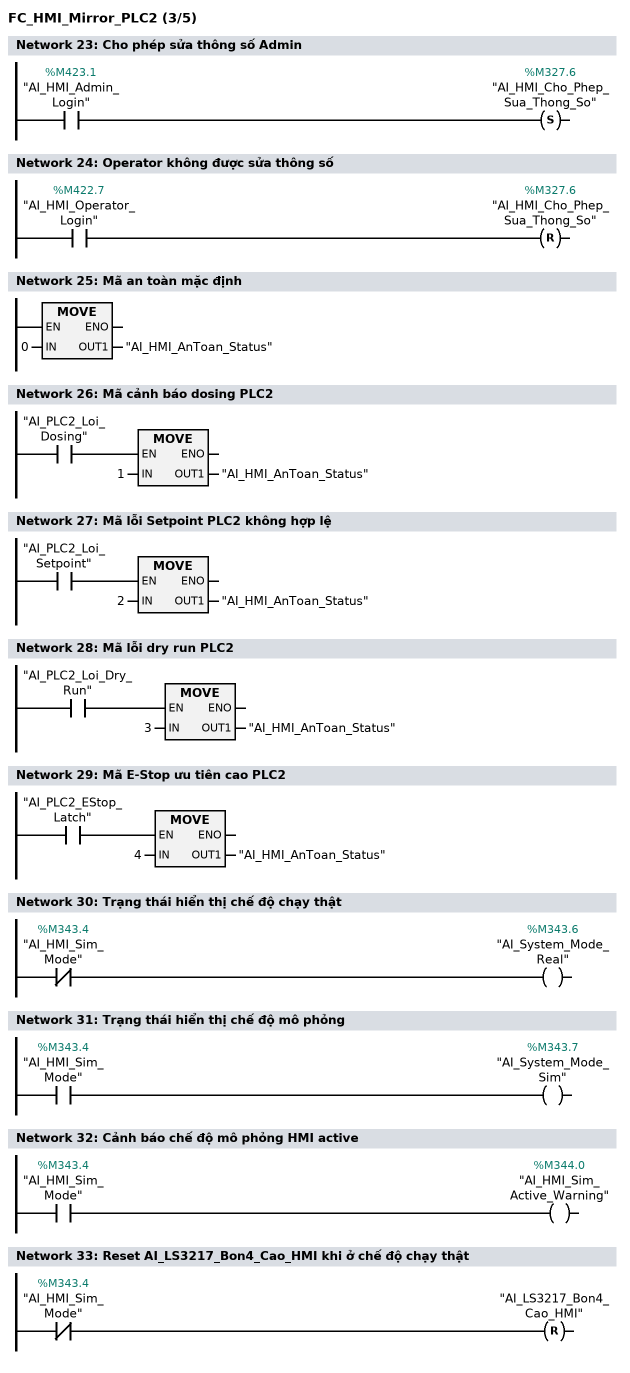
   RUNG wire#powerrail
      Contact( "AI_HMI_Admin_Login" )
      S_Coil( "AI_HMI_Cho_Phep_Sua_Thong_So" )
   END_RUNG
   // the same network as SCL:
   IF "AI_HMI_Admin_Login" THEN "AI_HMI_Cho_Phep_Sua_Thong_So" := TRUE; END_IF;
END_REGION

REGION Network 24: Operator không được sửa thông số
   RUNG wire#powerrail
      Contact( "AI_HMI_Operator_Login" )
      R_Coil( "AI_HMI_Cho_Phep_Sua_Thong_So" )
   END_RUNG
   // the same network as SCL:
   IF "AI_HMI_Operator_Login" THEN "AI_HMI_Cho_Phep_Sua_Thong_So" := FALSE; END_IF;
END_REGION

REGION Network 25: Mã an toàn mặc định
   RUNG wire#powerrail
      { S7_GenerateENO := "TRUE" } Move(in := 0, out1 => "AI_HMI_AnToan_Status")
   END_RUNG
   // the same network as SCL:
   "AI_HMI_AnToan_Status" := 0;
END_REGION

REGION Network 26: Mã cảnh báo dosing PLC2
   RUNG wire#powerrail
      Contact( "AI_PLC2_Loi_Dosing" )
      { S7_GenerateENO := "TRUE" } Move(in := 1, out1 => "AI_HMI_AnToan_Status")
   END_RUNG
   // the same network as SCL:
   IF "AI_PLC2_Loi_Dosing" THEN "AI_HMI_AnToan_Status" := 1; END_IF;
END_REGION

REGION Network 27: Mã lỗi Setpoint PLC2 không hợp lệ
   RUNG wire#powerrail
      Contact( "AI_PLC2_Loi_Setpoint" )
      { S7_GenerateENO := "TRUE" } Move(in := 2, out1 => "AI_HMI_AnToan_Status")
   END_RUNG
   // the same network as SCL:
   IF "AI_PLC2_Loi_Setpoint" THEN "AI_HMI_AnToan_Status" := 2; END_IF;
END_REGION

REGION Network 28: Mã lỗi dry run PLC2
   RUNG wire#powerrail
      Contact( "AI_PLC2_Loi_Dry_Run" )
      { S7_GenerateENO := "TRUE" } Move(in := 3, out1 => "AI_HMI_AnToan_Status")
   END_RUNG
   // the same network as SCL:
   IF "AI_PLC2_Loi_Dry_Run" THEN "AI_HMI_AnToan_Status" := 3; END_IF;
END_REGION

REGION Network 29: Mã E-Stop ưu tiên cao PLC2
   RUNG wire#powerrail
      Contact( "AI_PLC2_EStop_Latch" )
      { S7_GenerateENO := "TRUE" } Move(in := 4, out1 => "AI_HMI_AnToan_Status")
   END_RUNG
   // the same network as SCL:
   IF "AI_PLC2_EStop_Latch" THEN "AI_HMI_AnToan_Status" := 4; END_IF;
END_REGION

REGION Network 30: Trạng thái hiển thị chế độ chạy thật
   RUNG wire#powerrail
      I_Contact( "AI_HMI_Sim_Mode" )
      Coil( "AI_System_Mode_Real" )
   END_RUNG
   // the same network as SCL:
   "AI_System_Mode_Real" := NOT "AI_HMI_Sim_Mode";
END_REGION

REGION Network 31: Trạng thái hiển thị chế độ mô phỏng
   RUNG wire#powerrail
      Contact( "AI_HMI_Sim_Mode" )
      Coil( "AI_System_Mode_Sim" )
   END_RUNG
   // the same network as SCL:
   "AI_System_Mode_Sim" := "AI_HMI_Sim_Mode";
END_REGION

REGION Network 32: Cảnh báo chế độ mô phỏng HMI active
   RUNG wire#powerrail
      Contact( "AI_HMI_Sim_Mode" )
      Coil( "AI_HMI_Sim_Active_Warning" )
   END_RUNG
   // the same network as SCL:
   "AI_HMI_Sim_Active_Warning" := "AI_HMI_Sim_Mode";
END_REGION

REGION Network 33: Reset AI_LS3217_Bon4_Cao_HMI khi ở chế độ chạy thật
   RUNG wire#powerrail
      I_Contact( "AI_HMI_Sim_Mode" )
      R_Coil( "AI_LS3217_Bon4_Cao_HMI" )
   END_RUNG
   // the same network as SCL:
   IF NOT "AI_HMI_Sim_Mode" THEN "AI_LS3217_Bon4_Cao_HMI" := FALSE; END_IF;
END_REGION

REGION Network 34: Reset AI_Pump3265_Chuyen_Nhanh2_Cmd_Nhan_HMI khi ở chế độ chạy thật
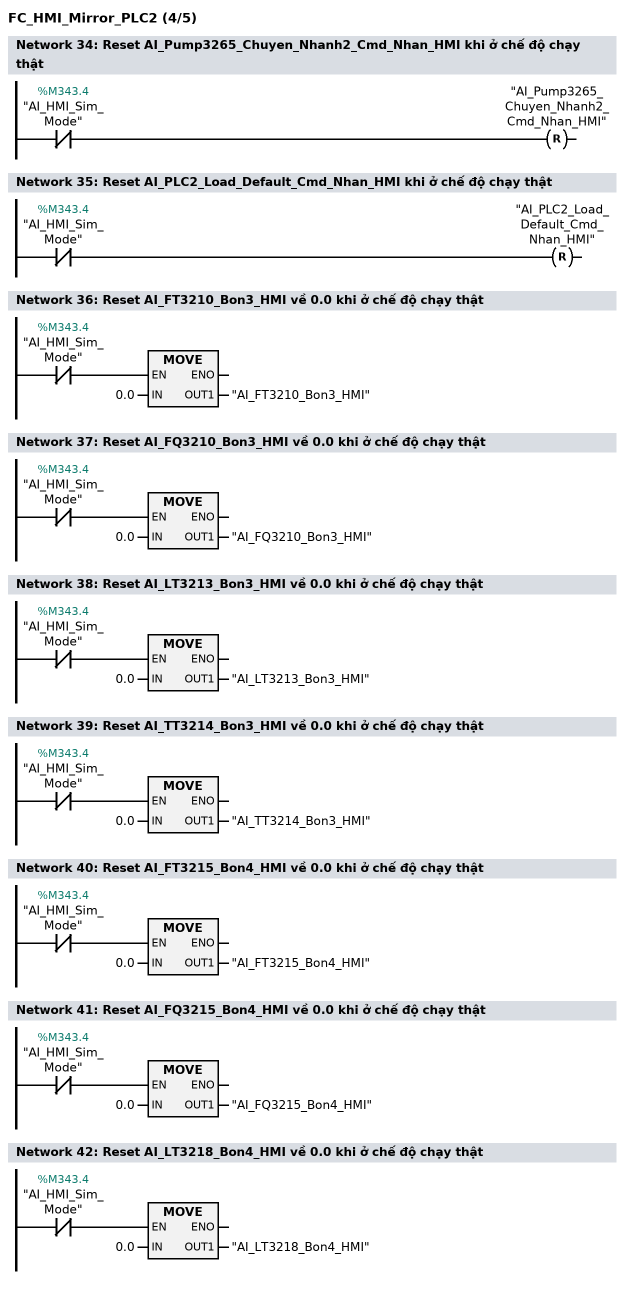
   RUNG wire#powerrail
      I_Contact( "AI_HMI_Sim_Mode" )
      R_Coil( "AI_Pump3265_Chuyen_Nhanh2_Cmd_Nhan_HMI" )
   END_RUNG
   // the same network as SCL:
   IF NOT "AI_HMI_Sim_Mode" THEN "AI_Pump3265_Chuyen_Nhanh2_Cmd_Nhan_HMI" := FALSE; END_IF;
END_REGION

REGION Network 35: Reset AI_PLC2_Load_Default_Cmd_Nhan_HMI khi ở chế độ chạy thật
   RUNG wire#powerrail
      I_Contact( "AI_HMI_Sim_Mode" )
      R_Coil( "AI_PLC2_Load_Default_Cmd_Nhan_HMI" )
   END_RUNG
   // the same network as SCL:
   IF NOT "AI_HMI_Sim_Mode" THEN "AI_PLC2_Load_Default_Cmd_Nhan_HMI" := FALSE; END_IF;
END_REGION

REGION Network 36: Reset AI_FT3210_Bon3_HMI về 0.0 khi ở chế độ chạy thật
   RUNG wire#powerrail
      I_Contact( "AI_HMI_Sim_Mode" )
      { S7_GenerateENO := "TRUE" } Move(in := 0.0, out1 => "AI_FT3210_Bon3_HMI")
   END_RUNG
   // the same network as SCL:
   IF NOT "AI_HMI_Sim_Mode" THEN "AI_FT3210_Bon3_HMI" := 0.0; END_IF;
END_REGION

REGION Network 37: Reset AI_FQ3210_Bon3_HMI về 0.0 khi ở chế độ chạy thật
   RUNG wire#powerrail
      I_Contact( "AI_HMI_Sim_Mode" )
      { S7_GenerateENO := "TRUE" } Move(in := 0.0, out1 => "AI_FQ3210_Bon3_HMI")
   END_RUNG
   // the same network as SCL:
   IF NOT "AI_HMI_Sim_Mode" THEN "AI_FQ3210_Bon3_HMI" := 0.0; END_IF;
END_REGION

REGION Network 38: Reset AI_LT3213_Bon3_HMI về 0.0 khi ở chế độ chạy thật
   RUNG wire#powerrail
      I_Contact( "AI_HMI_Sim_Mode" )
      { S7_GenerateENO := "TRUE" } Move(in := 0.0, out1 => "AI_LT3213_Bon3_HMI")
   END_RUNG
   // the same network as SCL:
   IF NOT "AI_HMI_Sim_Mode" THEN "AI_LT3213_Bon3_HMI" := 0.0; END_IF;
END_REGION

REGION Network 39: Reset AI_TT3214_Bon3_HMI về 0.0 khi ở chế độ chạy thật
   RUNG wire#powerrail
      I_Contact( "AI_HMI_Sim_Mode" )
      { S7_GenerateENO := "TRUE" } Move(in := 0.0, out1 => "AI_TT3214_Bon3_HMI")
   END_RUNG
   // the same network as SCL:
   IF NOT "AI_HMI_Sim_Mode" THEN "AI_TT3214_Bon3_HMI" := 0.0; END_IF;
END_REGION

REGION Network 40: Reset AI_FT3215_Bon4_HMI về 0.0 khi ở chế độ chạy thật
   RUNG wire#powerrail
      I_Contact( "AI_HMI_Sim_Mode" )
      { S7_GenerateENO := "TRUE" } Move(in := 0.0, out1 => "AI_FT3215_Bon4_HMI")
   END_RUNG
   // the same network as SCL:
   IF NOT "AI_HMI_Sim_Mode" THEN "AI_FT3215_Bon4_HMI" := 0.0; END_IF;
END_REGION

REGION Network 41: Reset AI_FQ3215_Bon4_HMI về 0.0 khi ở chế độ chạy thật
   RUNG wire#powerrail
      I_Contact( "AI_HMI_Sim_Mode" )
      { S7_GenerateENO := "TRUE" } Move(in := 0.0, out1 => "AI_FQ3215_Bon4_HMI")
   END_RUNG
   // the same network as SCL:
   IF NOT "AI_HMI_Sim_Mode" THEN "AI_FQ3215_Bon4_HMI" := 0.0; END_IF;
END_REGION

REGION Network 42: Reset AI_LT3218_Bon4_HMI về 0.0 khi ở chế độ chạy thật
   RUNG wire#powerrail
      I_Contact( "AI_HMI_Sim_Mode" )
      { S7_GenerateENO := "TRUE" } Move(in := 0.0, out1 => "AI_LT3218_Bon4_HMI")
   END_RUNG
   // the same network as SCL:
   IF NOT "AI_HMI_Sim_Mode" THEN "AI_LT3218_Bon4_HMI" := 0.0; END_IF;
END_REGION

REGION Network 43: Reset AI_TT3219_Bon4_HMI về 0.0 khi ở chế độ chạy thật
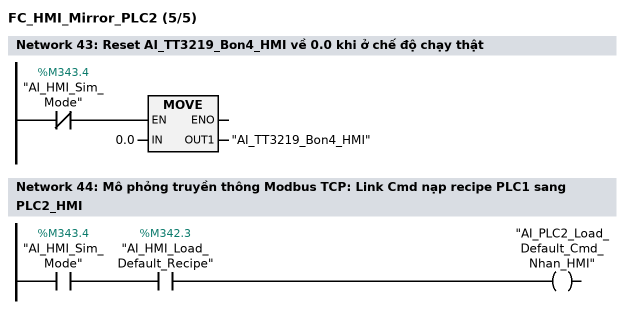
   RUNG wire#powerrail
      I_Contact( "AI_HMI_Sim_Mode" )
      { S7_GenerateENO := "TRUE" } Move(in := 0.0, out1 => "AI_TT3219_Bon4_HMI")
   END_RUNG
   // the same network as SCL:
   IF NOT "AI_HMI_Sim_Mode" THEN "AI_TT3219_Bon4_HMI" := 0.0; END_IF;
END_REGION

REGION Network 44: Mô phỏng truyền thông Modbus TCP: Link Cmd nạp recipe PLC1 sang PLC2_HMI
   RUNG wire#powerrail
      Contact( "AI_HMI_Sim_Mode" )
      Contact( "AI_HMI_Load_Default_Recipe" )
      Coil( "AI_PLC2_Load_Default_Cmd_Nhan_HMI" )
   END_RUNG
   // the same network as SCL:
   "AI_PLC2_Load_Default_Cmd_Nhan_HMI" := "AI_HMI_Sim_Mode" AND "AI_HMI_Load_Default_Recipe";
END_REGION
END_FUNCTION

FUNCTION "FC_Init_Default_Recipe_PLC2" : Void   // FC51, LAD
{ S7_Optimized_Access := 'TRUE' }
VERSION : 0.1
// stored: AutoNumber true, IsIECCheckEnabled false
BEGIN

REGION Network 1: Kích hoạt nạp recipe mặc định lần đầu scan PLC2
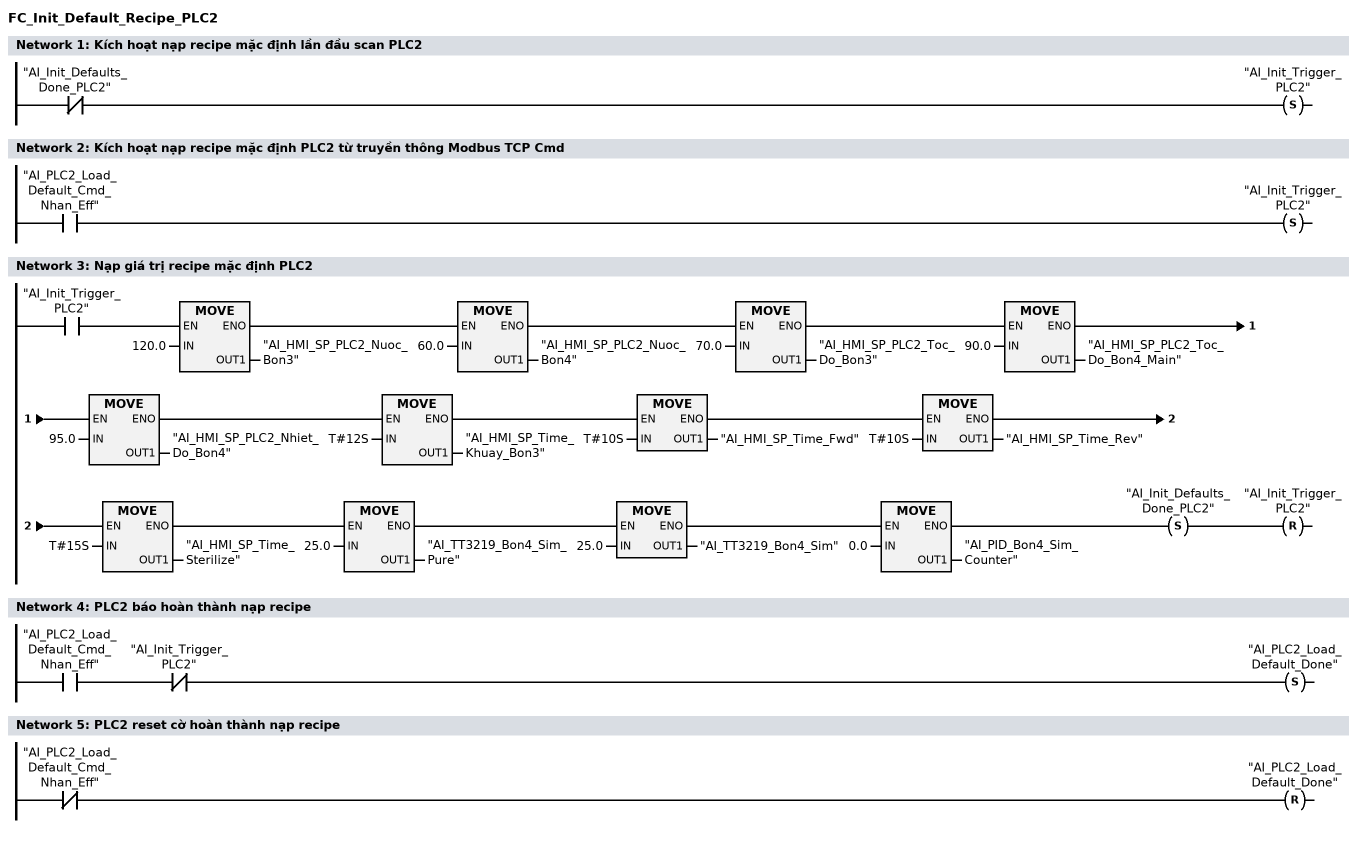
   RUNG wire#powerrail
      I_Contact( "AI_Init_Defaults_Done_PLC2" )
      S_Coil( "AI_Init_Trigger_PLC2" )
   END_RUNG
   // the same network as SCL:
   IF NOT "AI_Init_Defaults_Done_PLC2" THEN "AI_Init_Trigger_PLC2" := TRUE; END_IF;
END_REGION

REGION Network 2: Kích hoạt nạp recipe mặc định PLC2 từ truyền thông Modbus TCP Cmd
   RUNG wire#powerrail
      Contact( "AI_PLC2_Load_Default_Cmd_Nhan_Eff" )
      S_Coil( "AI_Init_Trigger_PLC2" )
   END_RUNG
   // the same network as SCL:
   IF "AI_PLC2_Load_Default_Cmd_Nhan_Eff" THEN "AI_Init_Trigger_PLC2" := TRUE; END_IF;
END_REGION

REGION Network 3: Nạp giá trị recipe mặc định PLC2
   RUNG wire#powerrail
      Contact( "AI_Init_Trigger_PLC2" )
      { S7_GenerateENO := "TRUE" } Move(in := 120.0, out1 => "AI_HMI_SP_PLC2_Nuoc_Bon3")
      { S7_GenerateENO := "TRUE" } Move(in := 60.0, out1 => "AI_HMI_SP_PLC2_Nuoc_Bon4")
      { S7_GenerateENO := "TRUE" } Move(in := 70.0, out1 => "AI_HMI_SP_PLC2_Toc_Do_Bon3")
      { S7_GenerateENO := "TRUE" } Move(in := 90.0, out1 => "AI_HMI_SP_PLC2_Toc_Do_Bon4_Main")
      { S7_GenerateENO := "TRUE" } Move(in := 95.0, out1 => "AI_HMI_SP_PLC2_Nhiet_Do_Bon4")
      { S7_GenerateENO := "TRUE" } Move(in := T#12S, out1 => "AI_HMI_SP_Time_Khuay_Bon3")
      { S7_GenerateENO := "TRUE" } Move(in := T#10S, out1 => "AI_HMI_SP_Time_Fwd")
      { S7_GenerateENO := "TRUE" } Move(in := T#10S, out1 => "AI_HMI_SP_Time_Rev")
      { S7_GenerateENO := "TRUE" } Move(in := T#15S, out1 => "AI_HMI_SP_Time_Sterilize")
      { S7_GenerateENO := "TRUE" } Move(in := 25.0, out1 => "AI_TT3219_Bon4_Sim_Pure")
      { S7_GenerateENO := "TRUE" } Move(in := 25.0, out1 => "AI_TT3219_Bon4_Sim")
      { S7_GenerateENO := "TRUE" } Move(in := 0.0, out1 => "AI_PID_Bon4_Sim_Counter")
      S_Coil( "AI_Init_Defaults_Done_PLC2" )
      R_Coil( "AI_Init_Trigger_PLC2" )
   END_RUNG
   // the same network as SCL:
   // ENO of a box is taken as its EN; it also drops when the box reports an error
   IF "AI_Init_Trigger_PLC2" THEN
       "AI_HMI_SP_PLC2_Nuoc_Bon3" := 120.0;
       "AI_HMI_SP_PLC2_Nuoc_Bon4" := 60.0;
       "AI_HMI_SP_PLC2_Toc_Do_Bon3" := 70.0;
       "AI_HMI_SP_PLC2_Toc_Do_Bon4_Main" := 90.0;
       "AI_HMI_SP_PLC2_Nhiet_Do_Bon4" := 95.0;
       "AI_HMI_SP_Time_Khuay_Bon3" := T#12S;
       "AI_HMI_SP_Time_Fwd" := T#10S;
       "AI_HMI_SP_Time_Rev" := T#10S;
       "AI_HMI_SP_Time_Sterilize" := T#15S;
       "AI_TT3219_Bon4_Sim_Pure" := 25.0;
       "AI_TT3219_Bon4_Sim" := 25.0;
       "AI_PID_Bon4_Sim_Counter" := 0.0;
       "AI_Init_Defaults_Done_PLC2" := TRUE;
       "AI_Init_Trigger_PLC2" := FALSE;
   END_IF;
END_REGION

REGION Network 4: PLC2 báo hoàn thành nạp recipe
   RUNG wire#powerrail
      Contact( "AI_PLC2_Load_Default_Cmd_Nhan_Eff" )
      I_Contact( "AI_Init_Trigger_PLC2" )
      S_Coil( "AI_PLC2_Load_Default_Done" )
   END_RUNG
   // the same network as SCL:
   IF "AI_PLC2_Load_Default_Cmd_Nhan_Eff" AND NOT "AI_Init_Trigger_PLC2" THEN
       "AI_PLC2_Load_Default_Done" := TRUE;
   END_IF;
END_REGION

REGION Network 5: PLC2 reset cờ hoàn thành nạp recipe
   RUNG wire#powerrail
      I_Contact( "AI_PLC2_Load_Default_Cmd_Nhan_Eff" )
      R_Coil( "AI_PLC2_Load_Default_Done" )
   END_RUNG
   // the same network as SCL:
   IF NOT "AI_PLC2_Load_Default_Cmd_Nhan_Eff" THEN "AI_PLC2_Load_Default_Done" := FALSE; END_IF;
END_REGION
END_FUNCTION

FUNCTION "FC_PLC2_Mixing" : Void   // FC20, LAD
{ S7_Optimized_Access := 'TRUE' }
VERSION : 0.1
// stored: AutoNumber true, IsIECCheckEnabled false
   VAR_TEMP   // added for the SCL form of the ladder/FBD networks
      _w1 : Bool;
   END_VAR
BEGIN

REGION Network 1: Khóa nút nhấn Start HMI qua Run Enable PLC2
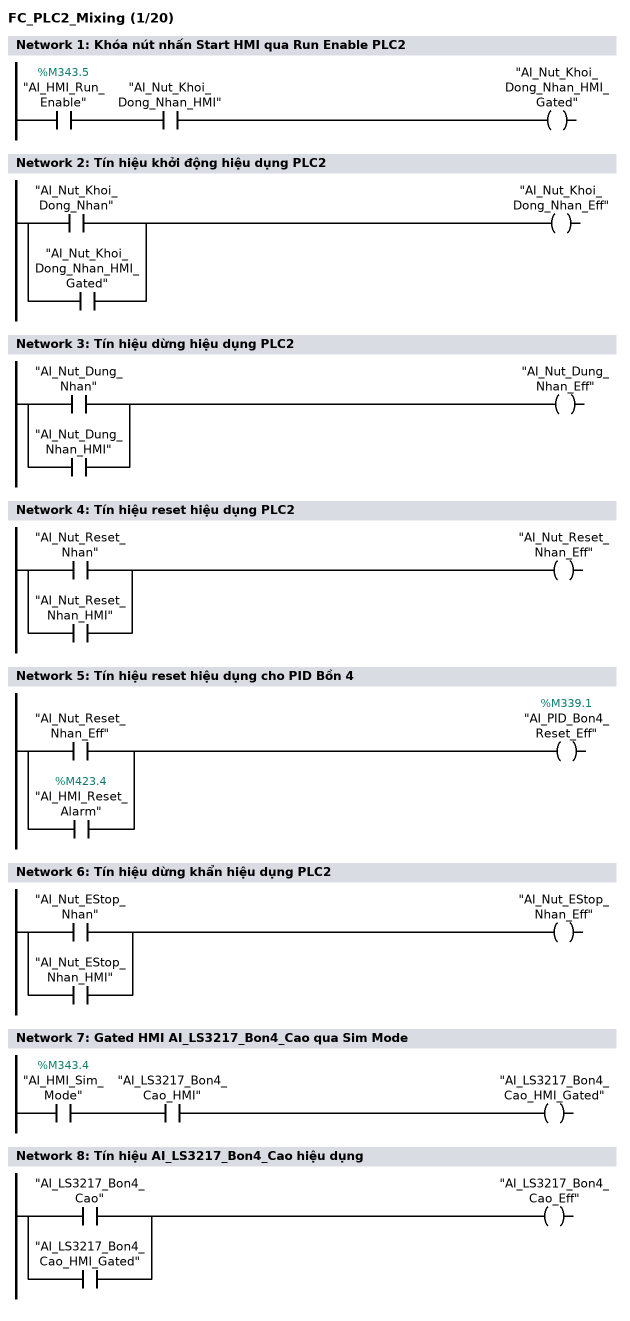
   RUNG wire#powerrail
      Contact( "AI_HMI_Run_Enable" )
      Contact( "AI_Nut_Khoi_Dong_Nhan_HMI" )
      Coil( "AI_Nut_Khoi_Dong_Nhan_HMI_Gated" )
   END_RUNG
   // the same network as SCL:
   "AI_Nut_Khoi_Dong_Nhan_HMI_Gated" := "AI_HMI_Run_Enable" AND "AI_Nut_Khoi_Dong_Nhan_HMI";
END_REGION

REGION Network 2: Tín hiệu khởi động hiệu dụng PLC2
   RUNG wire#powerrail
      Contact( "AI_Nut_Khoi_Dong_Nhan" )
      wire#w1
      Coil( "AI_Nut_Khoi_Dong_Nhan_Eff" )
   END_RUNG
   RUNG wire#powerrail
      Contact( "AI_Nut_Khoi_Dong_Nhan_HMI_Gated" )
   END_RUNG wire#w1
   // the same network as SCL:
   "AI_Nut_Khoi_Dong_Nhan_Eff" := "AI_Nut_Khoi_Dong_Nhan" OR "AI_Nut_Khoi_Dong_Nhan_HMI_Gated";
END_REGION

REGION Network 3: Tín hiệu dừng hiệu dụng PLC2
   RUNG wire#powerrail
      Contact( "AI_Nut_Dung_Nhan" )
      wire#w1
      Coil( "AI_Nut_Dung_Nhan_Eff" )
   END_RUNG
   RUNG wire#powerrail
      Contact( "AI_Nut_Dung_Nhan_HMI" )
   END_RUNG wire#w1
   // the same network as SCL:
   "AI_Nut_Dung_Nhan_Eff" := "AI_Nut_Dung_Nhan" OR "AI_Nut_Dung_Nhan_HMI";
END_REGION

REGION Network 4: Tín hiệu reset hiệu dụng PLC2
   RUNG wire#powerrail
      Contact( "AI_Nut_Reset_Nhan" )
      wire#w1
      Coil( "AI_Nut_Reset_Nhan_Eff" )
   END_RUNG
   RUNG wire#powerrail
      Contact( "AI_Nut_Reset_Nhan_HMI" )
   END_RUNG wire#w1
   // the same network as SCL:
   "AI_Nut_Reset_Nhan_Eff" := "AI_Nut_Reset_Nhan" OR "AI_Nut_Reset_Nhan_HMI";
END_REGION

REGION Network 5: Tín hiệu reset hiệu dụng cho PID Bồn 4
   RUNG wire#powerrail
      Contact( "AI_Nut_Reset_Nhan_Eff" )
      wire#w1
      Coil( "AI_PID_Bon4_Reset_Eff" )
   END_RUNG
   RUNG wire#powerrail
      Contact( "AI_HMI_Reset_Alarm" )
   END_RUNG wire#w1
   // the same network as SCL:
   "AI_PID_Bon4_Reset_Eff" := "AI_Nut_Reset_Nhan_Eff" OR "AI_HMI_Reset_Alarm";
END_REGION

REGION Network 6: Tín hiệu dừng khẩn hiệu dụng PLC2
   RUNG wire#powerrail
      Contact( "AI_Nut_EStop_Nhan" )
      wire#w1
      Coil( "AI_Nut_EStop_Nhan_Eff" )
   END_RUNG
   RUNG wire#powerrail
      Contact( "AI_Nut_EStop_Nhan_HMI" )
   END_RUNG wire#w1
   // the same network as SCL:
   "AI_Nut_EStop_Nhan_Eff" := "AI_Nut_EStop_Nhan" OR "AI_Nut_EStop_Nhan_HMI";
END_REGION

REGION Network 7: Gated HMI AI_LS3217_Bon4_Cao qua Sim Mode
   RUNG wire#powerrail
      Contact( "AI_HMI_Sim_Mode" )
      Contact( "AI_LS3217_Bon4_Cao_HMI" )
      Coil( "AI_LS3217_Bon4_Cao_HMI_Gated" )
   END_RUNG
   // the same network as SCL:
   "AI_LS3217_Bon4_Cao_HMI_Gated" := "AI_HMI_Sim_Mode" AND "AI_LS3217_Bon4_Cao_HMI";
END_REGION

REGION Network 8: Tín hiệu AI_LS3217_Bon4_Cao hiệu dụng
   RUNG wire#powerrail
      Contact( "AI_LS3217_Bon4_Cao" )
      wire#w1
      Coil( "AI_LS3217_Bon4_Cao_Eff" )
   END_RUNG
   RUNG wire#powerrail
      Contact( "AI_LS3217_Bon4_Cao_HMI_Gated" )
   END_RUNG wire#w1
   // the same network as SCL:
   "AI_LS3217_Bon4_Cao_Eff" := "AI_LS3217_Bon4_Cao" OR "AI_LS3217_Bon4_Cao_HMI_Gated";
END_REGION

REGION Network 9: Gated HMI AI_Pump3265_Chuyen_Nhanh2_Cmd_Nhan qua Sim Mode
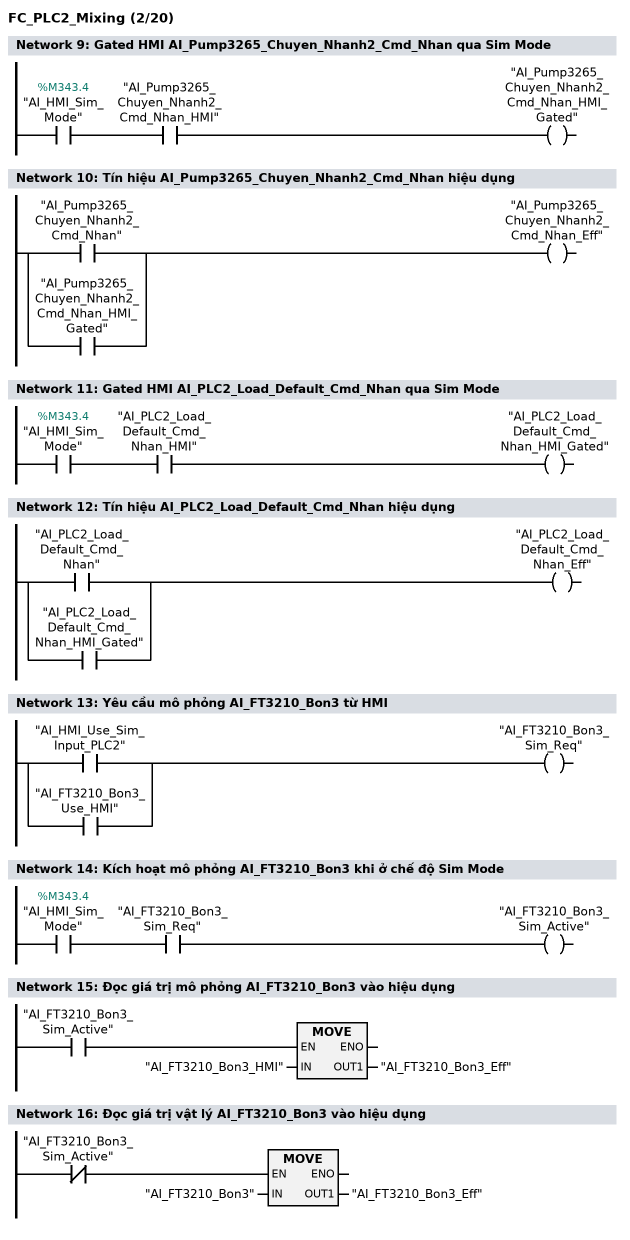
   RUNG wire#powerrail
      Contact( "AI_HMI_Sim_Mode" )
      Contact( "AI_Pump3265_Chuyen_Nhanh2_Cmd_Nhan_HMI" )
      Coil( "AI_Pump3265_Chuyen_Nhanh2_Cmd_Nhan_HMI_Gated" )
   END_RUNG
   // the same network as SCL:
   "AI_Pump3265_Chuyen_Nhanh2_Cmd_Nhan_HMI_Gated" := "AI_HMI_Sim_Mode" AND "AI_Pump3265_Chuyen_Nhanh2_Cmd_Nhan_HMI";
END_REGION

REGION Network 10: Tín hiệu AI_Pump3265_Chuyen_Nhanh2_Cmd_Nhan hiệu dụng
   RUNG wire#powerrail
      Contact( "AI_Pump3265_Chuyen_Nhanh2_Cmd_Nhan" )
      wire#w1
      Coil( "AI_Pump3265_Chuyen_Nhanh2_Cmd_Nhan_Eff" )
   END_RUNG
   RUNG wire#powerrail
      Contact( "AI_Pump3265_Chuyen_Nhanh2_Cmd_Nhan_HMI_Gated" )
   END_RUNG wire#w1
   // the same network as SCL:
   "AI_Pump3265_Chuyen_Nhanh2_Cmd_Nhan_Eff" := "AI_Pump3265_Chuyen_Nhanh2_Cmd_Nhan" OR "AI_Pump3265_Chuyen_Nhanh2_Cmd_Nhan_HMI_Gated";
END_REGION

REGION Network 11: Gated HMI AI_PLC2_Load_Default_Cmd_Nhan qua Sim Mode
   RUNG wire#powerrail
      Contact( "AI_HMI_Sim_Mode" )
      Contact( "AI_PLC2_Load_Default_Cmd_Nhan_HMI" )
      Coil( "AI_PLC2_Load_Default_Cmd_Nhan_HMI_Gated" )
   END_RUNG
   // the same network as SCL:
   "AI_PLC2_Load_Default_Cmd_Nhan_HMI_Gated" := "AI_HMI_Sim_Mode" AND "AI_PLC2_Load_Default_Cmd_Nhan_HMI";
END_REGION

REGION Network 12: Tín hiệu AI_PLC2_Load_Default_Cmd_Nhan hiệu dụng
   RUNG wire#powerrail
      Contact( "AI_PLC2_Load_Default_Cmd_Nhan" )
      wire#w1
      Coil( "AI_PLC2_Load_Default_Cmd_Nhan_Eff" )
   END_RUNG
   RUNG wire#powerrail
      Contact( "AI_PLC2_Load_Default_Cmd_Nhan_HMI_Gated" )
   END_RUNG wire#w1
   // the same network as SCL:
   "AI_PLC2_Load_Default_Cmd_Nhan_Eff" := "AI_PLC2_Load_Default_Cmd_Nhan" OR "AI_PLC2_Load_Default_Cmd_Nhan_HMI_Gated";
END_REGION

REGION Network 13: Yêu cầu mô phỏng AI_FT3210_Bon3 từ HMI
   RUNG wire#powerrail
      Contact( "AI_HMI_Use_Sim_Input_PLC2" )
      wire#w1
      Coil( "AI_FT3210_Bon3_Sim_Req" )
   END_RUNG
   RUNG wire#powerrail
      Contact( "AI_FT3210_Bon3_Use_HMI" )
   END_RUNG wire#w1
   // the same network as SCL:
   "AI_FT3210_Bon3_Sim_Req" := "AI_HMI_Use_Sim_Input_PLC2" OR "AI_FT3210_Bon3_Use_HMI";
END_REGION

REGION Network 14: Kích hoạt mô phỏng AI_FT3210_Bon3 khi ở chế độ Sim Mode
   RUNG wire#powerrail
      Contact( "AI_HMI_Sim_Mode" )
      Contact( "AI_FT3210_Bon3_Sim_Req" )
      Coil( "AI_FT3210_Bon3_Sim_Active" )
   END_RUNG
   // the same network as SCL:
   "AI_FT3210_Bon3_Sim_Active" := "AI_HMI_Sim_Mode" AND "AI_FT3210_Bon3_Sim_Req";
END_REGION

REGION Network 15: Đọc giá trị mô phỏng AI_FT3210_Bon3 vào hiệu dụng
   RUNG wire#powerrail
      Contact( "AI_FT3210_Bon3_Sim_Active" )
      { S7_GenerateENO := "TRUE" } Move(in := "AI_FT3210_Bon3_HMI", out1 => "AI_FT3210_Bon3_Eff")
   END_RUNG
   // the same network as SCL:
   IF "AI_FT3210_Bon3_Sim_Active" THEN "AI_FT3210_Bon3_Eff" := "AI_FT3210_Bon3_HMI"; END_IF;
END_REGION

REGION Network 16: Đọc giá trị vật lý AI_FT3210_Bon3 vào hiệu dụng
   RUNG wire#powerrail
      I_Contact( "AI_FT3210_Bon3_Sim_Active" )
      { S7_GenerateENO := "TRUE" } Move(in := "AI_FT3210_Bon3", out1 => "AI_FT3210_Bon3_Eff")
   END_RUNG
   // the same network as SCL:
   IF NOT "AI_FT3210_Bon3_Sim_Active" THEN "AI_FT3210_Bon3_Eff" := "AI_FT3210_Bon3"; END_IF;
END_REGION

REGION Network 17: Yêu cầu mô phỏng AI_FQ3210_Bon3 từ HMI
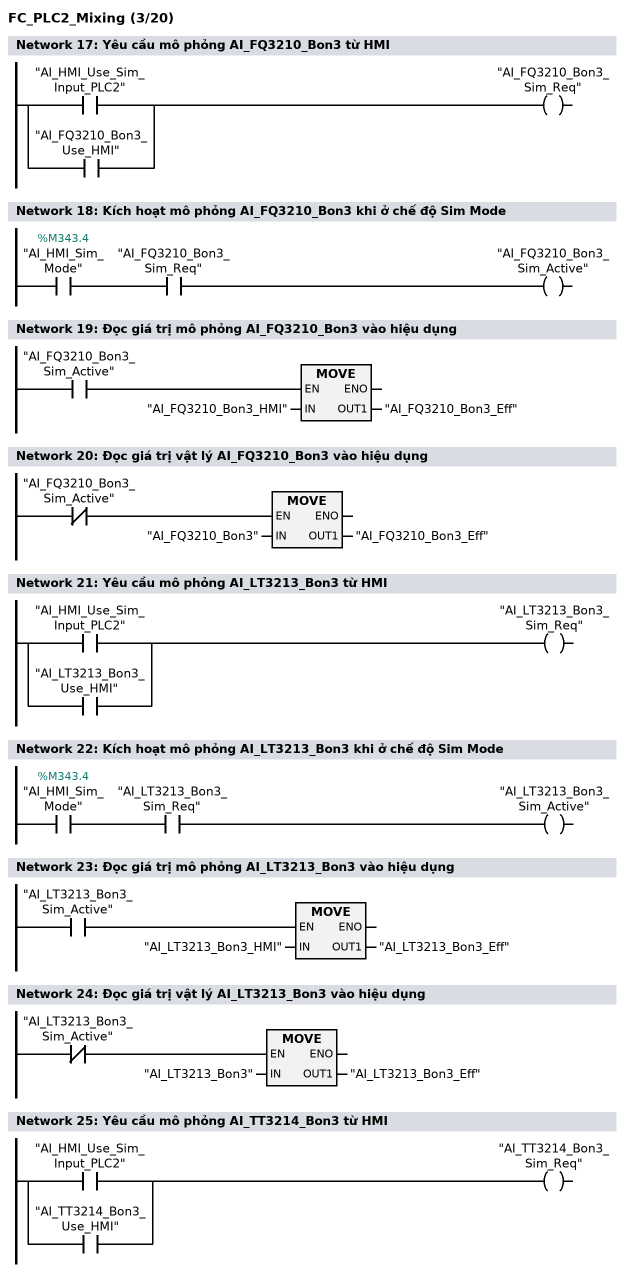
   RUNG wire#powerrail
      Contact( "AI_HMI_Use_Sim_Input_PLC2" )
      wire#w1
      Coil( "AI_FQ3210_Bon3_Sim_Req" )
   END_RUNG
   RUNG wire#powerrail
      Contact( "AI_FQ3210_Bon3_Use_HMI" )
   END_RUNG wire#w1
   // the same network as SCL:
   "AI_FQ3210_Bon3_Sim_Req" := "AI_HMI_Use_Sim_Input_PLC2" OR "AI_FQ3210_Bon3_Use_HMI";
END_REGION

REGION Network 18: Kích hoạt mô phỏng AI_FQ3210_Bon3 khi ở chế độ Sim Mode
   RUNG wire#powerrail
      Contact( "AI_HMI_Sim_Mode" )
      Contact( "AI_FQ3210_Bon3_Sim_Req" )
      Coil( "AI_FQ3210_Bon3_Sim_Active" )
   END_RUNG
   // the same network as SCL:
   "AI_FQ3210_Bon3_Sim_Active" := "AI_HMI_Sim_Mode" AND "AI_FQ3210_Bon3_Sim_Req";
END_REGION

REGION Network 19: Đọc giá trị mô phỏng AI_FQ3210_Bon3 vào hiệu dụng
   RUNG wire#powerrail
      Contact( "AI_FQ3210_Bon3_Sim_Active" )
      { S7_GenerateENO := "TRUE" } Move(in := "AI_FQ3210_Bon3_HMI", out1 => "AI_FQ3210_Bon3_Eff")
   END_RUNG
   // the same network as SCL:
   IF "AI_FQ3210_Bon3_Sim_Active" THEN "AI_FQ3210_Bon3_Eff" := "AI_FQ3210_Bon3_HMI"; END_IF;
END_REGION

REGION Network 20: Đọc giá trị vật lý AI_FQ3210_Bon3 vào hiệu dụng
   RUNG wire#powerrail
      I_Contact( "AI_FQ3210_Bon3_Sim_Active" )
      { S7_GenerateENO := "TRUE" } Move(in := "AI_FQ3210_Bon3", out1 => "AI_FQ3210_Bon3_Eff")
   END_RUNG
   // the same network as SCL:
   IF NOT "AI_FQ3210_Bon3_Sim_Active" THEN "AI_FQ3210_Bon3_Eff" := "AI_FQ3210_Bon3"; END_IF;
END_REGION

REGION Network 21: Yêu cầu mô phỏng AI_LT3213_Bon3 từ HMI
   RUNG wire#powerrail
      Contact( "AI_HMI_Use_Sim_Input_PLC2" )
      wire#w1
      Coil( "AI_LT3213_Bon3_Sim_Req" )
   END_RUNG
   RUNG wire#powerrail
      Contact( "AI_LT3213_Bon3_Use_HMI" )
   END_RUNG wire#w1
   // the same network as SCL:
   "AI_LT3213_Bon3_Sim_Req" := "AI_HMI_Use_Sim_Input_PLC2" OR "AI_LT3213_Bon3_Use_HMI";
END_REGION

REGION Network 22: Kích hoạt mô phỏng AI_LT3213_Bon3 khi ở chế độ Sim Mode
   RUNG wire#powerrail
      Contact( "AI_HMI_Sim_Mode" )
      Contact( "AI_LT3213_Bon3_Sim_Req" )
      Coil( "AI_LT3213_Bon3_Sim_Active" )
   END_RUNG
   // the same network as SCL:
   "AI_LT3213_Bon3_Sim_Active" := "AI_HMI_Sim_Mode" AND "AI_LT3213_Bon3_Sim_Req";
END_REGION

REGION Network 23: Đọc giá trị mô phỏng AI_LT3213_Bon3 vào hiệu dụng
   RUNG wire#powerrail
      Contact( "AI_LT3213_Bon3_Sim_Active" )
      { S7_GenerateENO := "TRUE" } Move(in := "AI_LT3213_Bon3_HMI", out1 => "AI_LT3213_Bon3_Eff")
   END_RUNG
   // the same network as SCL:
   IF "AI_LT3213_Bon3_Sim_Active" THEN "AI_LT3213_Bon3_Eff" := "AI_LT3213_Bon3_HMI"; END_IF;
END_REGION

REGION Network 24: Đọc giá trị vật lý AI_LT3213_Bon3 vào hiệu dụng
   RUNG wire#powerrail
      I_Contact( "AI_LT3213_Bon3_Sim_Active" )
      { S7_GenerateENO := "TRUE" } Move(in := "AI_LT3213_Bon3", out1 => "AI_LT3213_Bon3_Eff")
   END_RUNG
   // the same network as SCL:
   IF NOT "AI_LT3213_Bon3_Sim_Active" THEN "AI_LT3213_Bon3_Eff" := "AI_LT3213_Bon3"; END_IF;
END_REGION

REGION Network 25: Yêu cầu mô phỏng AI_TT3214_Bon3 từ HMI
   RUNG wire#powerrail
      Contact( "AI_HMI_Use_Sim_Input_PLC2" )
      wire#w1
      Coil( "AI_TT3214_Bon3_Sim_Req" )
   END_RUNG
   RUNG wire#powerrail
      Contact( "AI_TT3214_Bon3_Use_HMI" )
   END_RUNG wire#w1
   // the same network as SCL:
   "AI_TT3214_Bon3_Sim_Req" := "AI_HMI_Use_Sim_Input_PLC2" OR "AI_TT3214_Bon3_Use_HMI";
END_REGION

REGION Network 26: Kích hoạt mô phỏng AI_TT3214_Bon3 khi ở chế độ Sim Mode
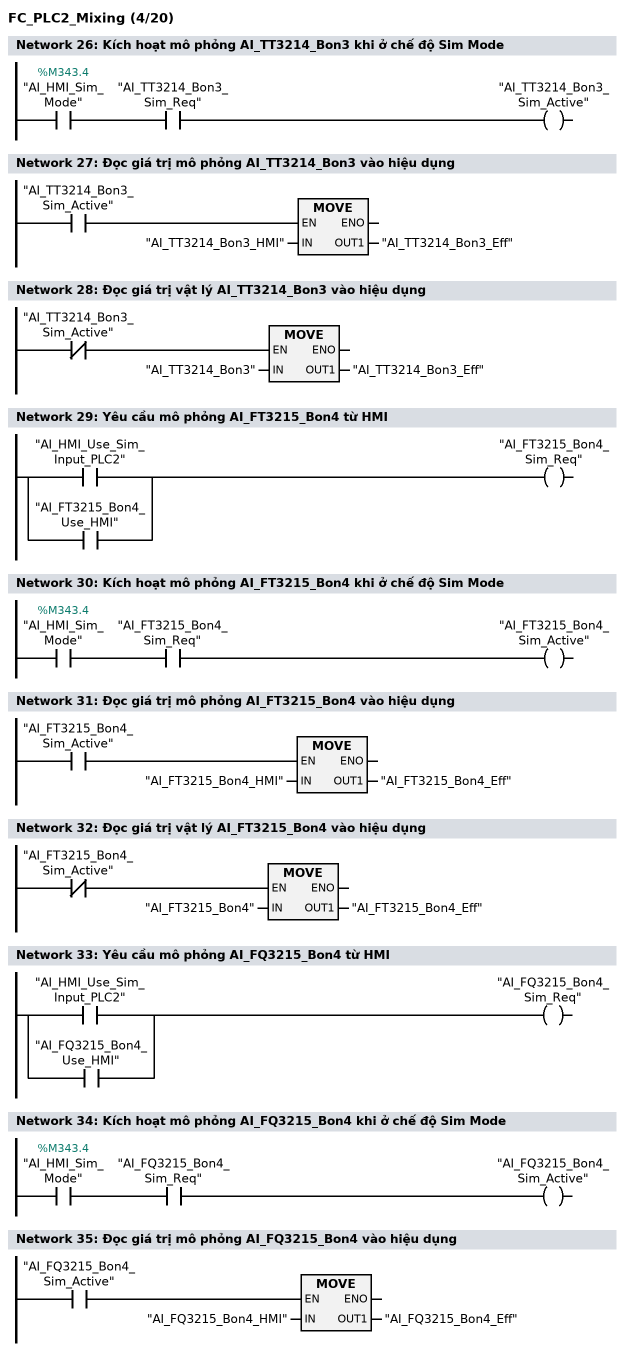
   RUNG wire#powerrail
      Contact( "AI_HMI_Sim_Mode" )
      Contact( "AI_TT3214_Bon3_Sim_Req" )
      Coil( "AI_TT3214_Bon3_Sim_Active" )
   END_RUNG
   // the same network as SCL:
   "AI_TT3214_Bon3_Sim_Active" := "AI_HMI_Sim_Mode" AND "AI_TT3214_Bon3_Sim_Req";
END_REGION

REGION Network 27: Đọc giá trị mô phỏng AI_TT3214_Bon3 vào hiệu dụng
   RUNG wire#powerrail
      Contact( "AI_TT3214_Bon3_Sim_Active" )
      { S7_GenerateENO := "TRUE" } Move(in := "AI_TT3214_Bon3_HMI", out1 => "AI_TT3214_Bon3_Eff")
   END_RUNG
   // the same network as SCL:
   IF "AI_TT3214_Bon3_Sim_Active" THEN "AI_TT3214_Bon3_Eff" := "AI_TT3214_Bon3_HMI"; END_IF;
END_REGION

REGION Network 28: Đọc giá trị vật lý AI_TT3214_Bon3 vào hiệu dụng
   RUNG wire#powerrail
      I_Contact( "AI_TT3214_Bon3_Sim_Active" )
      { S7_GenerateENO := "TRUE" } Move(in := "AI_TT3214_Bon3", out1 => "AI_TT3214_Bon3_Eff")
   END_RUNG
   // the same network as SCL:
   IF NOT "AI_TT3214_Bon3_Sim_Active" THEN "AI_TT3214_Bon3_Eff" := "AI_TT3214_Bon3"; END_IF;
END_REGION

REGION Network 29: Yêu cầu mô phỏng AI_FT3215_Bon4 từ HMI
   RUNG wire#powerrail
      Contact( "AI_HMI_Use_Sim_Input_PLC2" )
      wire#w1
      Coil( "AI_FT3215_Bon4_Sim_Req" )
   END_RUNG
   RUNG wire#powerrail
      Contact( "AI_FT3215_Bon4_Use_HMI" )
   END_RUNG wire#w1
   // the same network as SCL:
   "AI_FT3215_Bon4_Sim_Req" := "AI_HMI_Use_Sim_Input_PLC2" OR "AI_FT3215_Bon4_Use_HMI";
END_REGION

REGION Network 30: Kích hoạt mô phỏng AI_FT3215_Bon4 khi ở chế độ Sim Mode
   RUNG wire#powerrail
      Contact( "AI_HMI_Sim_Mode" )
      Contact( "AI_FT3215_Bon4_Sim_Req" )
      Coil( "AI_FT3215_Bon4_Sim_Active" )
   END_RUNG
   // the same network as SCL:
   "AI_FT3215_Bon4_Sim_Active" := "AI_HMI_Sim_Mode" AND "AI_FT3215_Bon4_Sim_Req";
END_REGION

REGION Network 31: Đọc giá trị mô phỏng AI_FT3215_Bon4 vào hiệu dụng
   RUNG wire#powerrail
      Contact( "AI_FT3215_Bon4_Sim_Active" )
      { S7_GenerateENO := "TRUE" } Move(in := "AI_FT3215_Bon4_HMI", out1 => "AI_FT3215_Bon4_Eff")
   END_RUNG
   // the same network as SCL:
   IF "AI_FT3215_Bon4_Sim_Active" THEN "AI_FT3215_Bon4_Eff" := "AI_FT3215_Bon4_HMI"; END_IF;
END_REGION

REGION Network 32: Đọc giá trị vật lý AI_FT3215_Bon4 vào hiệu dụng
   RUNG wire#powerrail
      I_Contact( "AI_FT3215_Bon4_Sim_Active" )
      { S7_GenerateENO := "TRUE" } Move(in := "AI_FT3215_Bon4", out1 => "AI_FT3215_Bon4_Eff")
   END_RUNG
   // the same network as SCL:
   IF NOT "AI_FT3215_Bon4_Sim_Active" THEN "AI_FT3215_Bon4_Eff" := "AI_FT3215_Bon4"; END_IF;
END_REGION

REGION Network 33: Yêu cầu mô phỏng AI_FQ3215_Bon4 từ HMI
   RUNG wire#powerrail
      Contact( "AI_HMI_Use_Sim_Input_PLC2" )
      wire#w1
      Coil( "AI_FQ3215_Bon4_Sim_Req" )
   END_RUNG
   RUNG wire#powerrail
      Contact( "AI_FQ3215_Bon4_Use_HMI" )
   END_RUNG wire#w1
   // the same network as SCL:
   "AI_FQ3215_Bon4_Sim_Req" := "AI_HMI_Use_Sim_Input_PLC2" OR "AI_FQ3215_Bon4_Use_HMI";
END_REGION

REGION Network 34: Kích hoạt mô phỏng AI_FQ3215_Bon4 khi ở chế độ Sim Mode
   RUNG wire#powerrail
      Contact( "AI_HMI_Sim_Mode" )
      Contact( "AI_FQ3215_Bon4_Sim_Req" )
      Coil( "AI_FQ3215_Bon4_Sim_Active" )
   END_RUNG
   // the same network as SCL:
   "AI_FQ3215_Bon4_Sim_Active" := "AI_HMI_Sim_Mode" AND "AI_FQ3215_Bon4_Sim_Req";
END_REGION

REGION Network 35: Đọc giá trị mô phỏng AI_FQ3215_Bon4 vào hiệu dụng
   RUNG wire#powerrail
      Contact( "AI_FQ3215_Bon4_Sim_Active" )
      { S7_GenerateENO := "TRUE" } Move(in := "AI_FQ3215_Bon4_HMI", out1 => "AI_FQ3215_Bon4_Eff")
   END_RUNG
   // the same network as SCL:
   IF "AI_FQ3215_Bon4_Sim_Active" THEN "AI_FQ3215_Bon4_Eff" := "AI_FQ3215_Bon4_HMI"; END_IF;
END_REGION

REGION Network 36: Đọc giá trị vật lý AI_FQ3215_Bon4 vào hiệu dụng
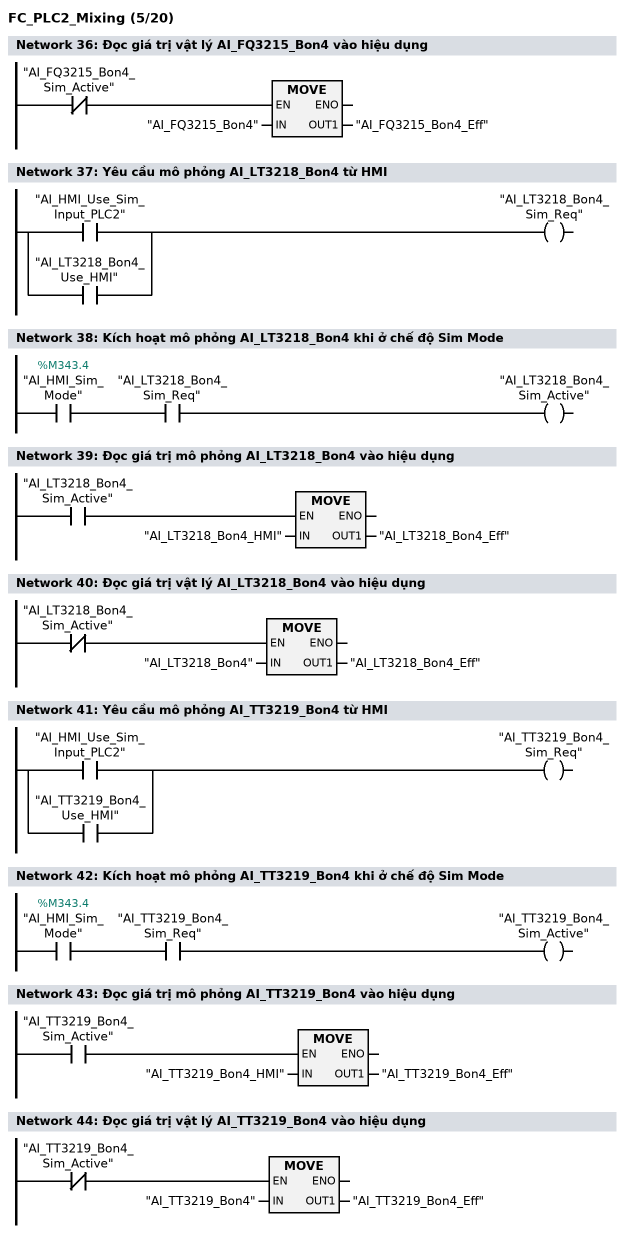
   RUNG wire#powerrail
      I_Contact( "AI_FQ3215_Bon4_Sim_Active" )
      { S7_GenerateENO := "TRUE" } Move(in := "AI_FQ3215_Bon4", out1 => "AI_FQ3215_Bon4_Eff")
   END_RUNG
   // the same network as SCL:
   IF NOT "AI_FQ3215_Bon4_Sim_Active" THEN "AI_FQ3215_Bon4_Eff" := "AI_FQ3215_Bon4"; END_IF;
END_REGION

REGION Network 37: Yêu cầu mô phỏng AI_LT3218_Bon4 từ HMI
   RUNG wire#powerrail
      Contact( "AI_HMI_Use_Sim_Input_PLC2" )
      wire#w1
      Coil( "AI_LT3218_Bon4_Sim_Req" )
   END_RUNG
   RUNG wire#powerrail
      Contact( "AI_LT3218_Bon4_Use_HMI" )
   END_RUNG wire#w1
   // the same network as SCL:
   "AI_LT3218_Bon4_Sim_Req" := "AI_HMI_Use_Sim_Input_PLC2" OR "AI_LT3218_Bon4_Use_HMI";
END_REGION

REGION Network 38: Kích hoạt mô phỏng AI_LT3218_Bon4 khi ở chế độ Sim Mode
   RUNG wire#powerrail
      Contact( "AI_HMI_Sim_Mode" )
      Contact( "AI_LT3218_Bon4_Sim_Req" )
      Coil( "AI_LT3218_Bon4_Sim_Active" )
   END_RUNG
   // the same network as SCL:
   "AI_LT3218_Bon4_Sim_Active" := "AI_HMI_Sim_Mode" AND "AI_LT3218_Bon4_Sim_Req";
END_REGION

REGION Network 39: Đọc giá trị mô phỏng AI_LT3218_Bon4 vào hiệu dụng
   RUNG wire#powerrail
      Contact( "AI_LT3218_Bon4_Sim_Active" )
      { S7_GenerateENO := "TRUE" } Move(in := "AI_LT3218_Bon4_HMI", out1 => "AI_LT3218_Bon4_Eff")
   END_RUNG
   // the same network as SCL:
   IF "AI_LT3218_Bon4_Sim_Active" THEN "AI_LT3218_Bon4_Eff" := "AI_LT3218_Bon4_HMI"; END_IF;
END_REGION

REGION Network 40: Đọc giá trị vật lý AI_LT3218_Bon4 vào hiệu dụng
   RUNG wire#powerrail
      I_Contact( "AI_LT3218_Bon4_Sim_Active" )
      { S7_GenerateENO := "TRUE" } Move(in := "AI_LT3218_Bon4", out1 => "AI_LT3218_Bon4_Eff")
   END_RUNG
   // the same network as SCL:
   IF NOT "AI_LT3218_Bon4_Sim_Active" THEN "AI_LT3218_Bon4_Eff" := "AI_LT3218_Bon4"; END_IF;
END_REGION

REGION Network 41: Yêu cầu mô phỏng AI_TT3219_Bon4 từ HMI
   RUNG wire#powerrail
      Contact( "AI_HMI_Use_Sim_Input_PLC2" )
      wire#w1
      Coil( "AI_TT3219_Bon4_Sim_Req" )
   END_RUNG
   RUNG wire#powerrail
      Contact( "AI_TT3219_Bon4_Use_HMI" )
   END_RUNG wire#w1
   // the same network as SCL:
   "AI_TT3219_Bon4_Sim_Req" := "AI_HMI_Use_Sim_Input_PLC2" OR "AI_TT3219_Bon4_Use_HMI";
END_REGION

REGION Network 42: Kích hoạt mô phỏng AI_TT3219_Bon4 khi ở chế độ Sim Mode
   RUNG wire#powerrail
      Contact( "AI_HMI_Sim_Mode" )
      Contact( "AI_TT3219_Bon4_Sim_Req" )
      Coil( "AI_TT3219_Bon4_Sim_Active" )
   END_RUNG
   // the same network as SCL:
   "AI_TT3219_Bon4_Sim_Active" := "AI_HMI_Sim_Mode" AND "AI_TT3219_Bon4_Sim_Req";
END_REGION

REGION Network 43: Đọc giá trị mô phỏng AI_TT3219_Bon4 vào hiệu dụng
   RUNG wire#powerrail
      Contact( "AI_TT3219_Bon4_Sim_Active" )
      { S7_GenerateENO := "TRUE" } Move(in := "AI_TT3219_Bon4_HMI", out1 => "AI_TT3219_Bon4_Eff")
   END_RUNG
   // the same network as SCL:
   IF "AI_TT3219_Bon4_Sim_Active" THEN "AI_TT3219_Bon4_Eff" := "AI_TT3219_Bon4_HMI"; END_IF;
END_REGION

REGION Network 44: Đọc giá trị vật lý AI_TT3219_Bon4 vào hiệu dụng
   RUNG wire#powerrail
      I_Contact( "AI_TT3219_Bon4_Sim_Active" )
      { S7_GenerateENO := "TRUE" } Move(in := "AI_TT3219_Bon4", out1 => "AI_TT3219_Bon4_Eff")
   END_RUNG
   // the same network as SCL:
   IF NOT "AI_TT3219_Bon4_Sim_Active" THEN "AI_TT3219_Bon4_Eff" := "AI_TT3219_Bon4"; END_IF;
END_REGION

REGION Network 45: Kiểm tra hợp lệ Setpoint PLC2
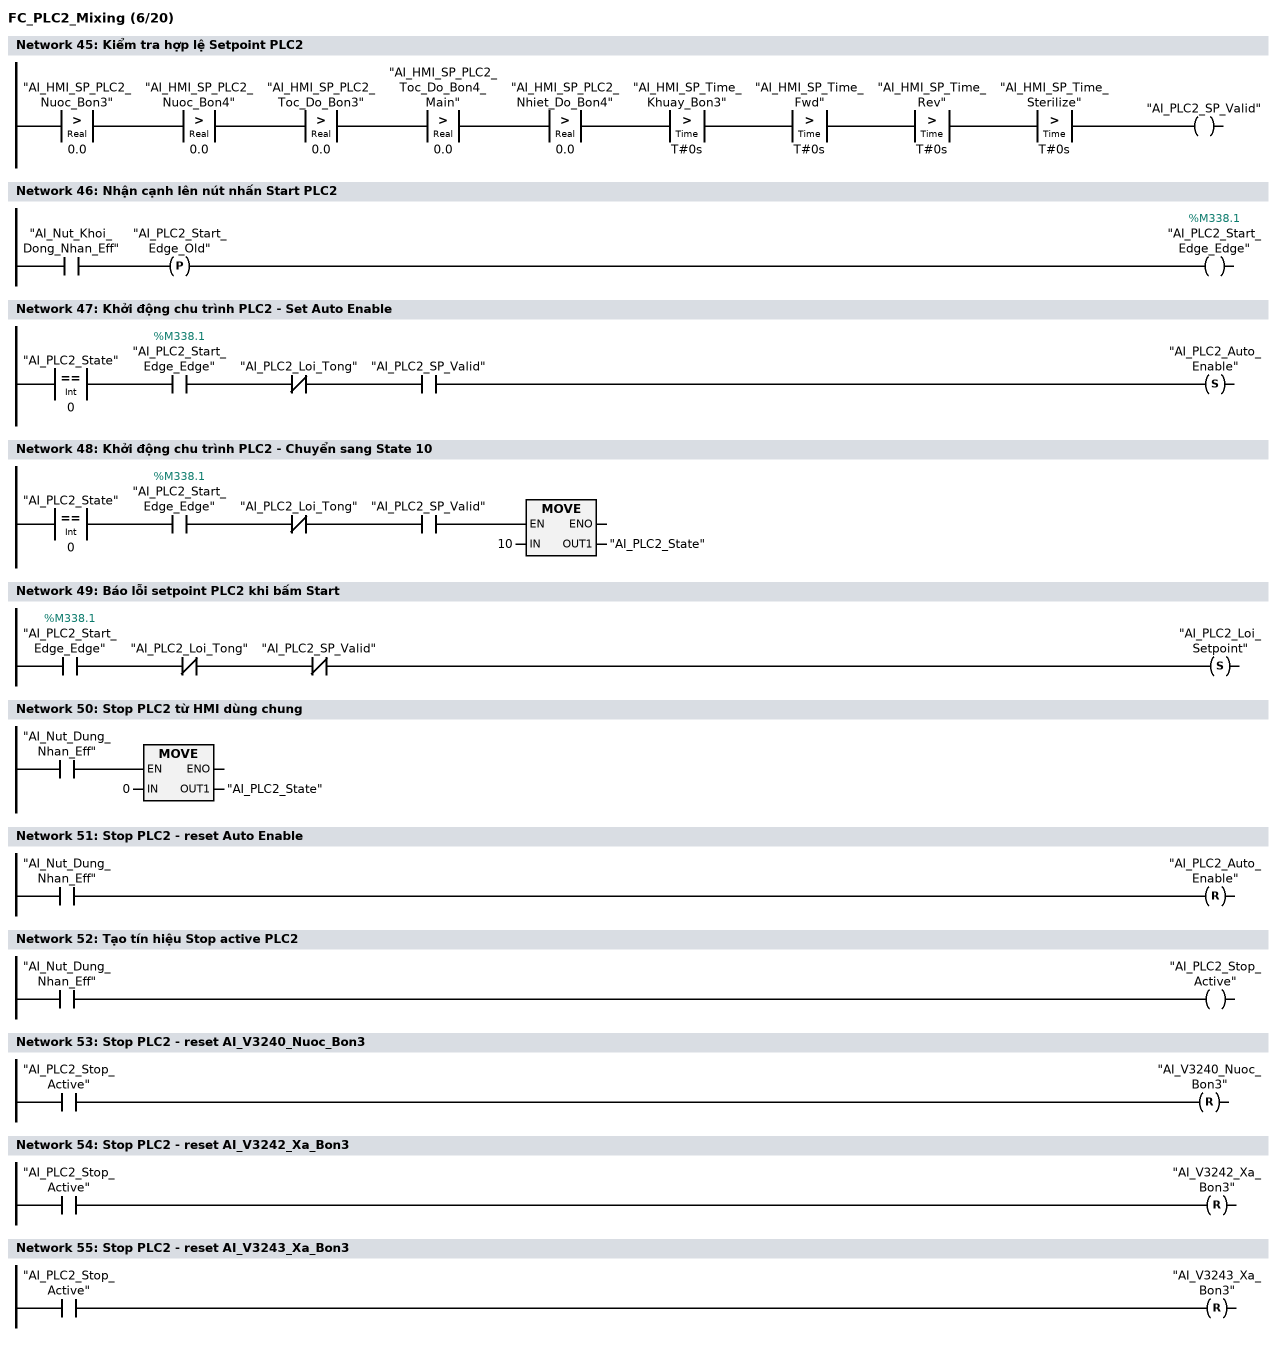
   RUNG wire#powerrail
      { S7_Templates := "SrcType := Real" } GT_Contact(in1 := "AI_HMI_SP_PLC2_Nuoc_Bon3", in2 := 0.0)
      { S7_Templates := "SrcType := Real" } GT_Contact(in1 := "AI_HMI_SP_PLC2_Nuoc_Bon4", in2 := 0.0)
      { S7_Templates := "SrcType := Real" } GT_Contact(in1 := "AI_HMI_SP_PLC2_Toc_Do_Bon3", in2 := 0.0)
      { S7_Templates := "SrcType := Real" } GT_Contact(in1 := "AI_HMI_SP_PLC2_Toc_Do_Bon4_Main", in2 := 0.0)
      { S7_Templates := "SrcType := Real" } GT_Contact(in1 := "AI_HMI_SP_PLC2_Nhiet_Do_Bon4", in2 := 0.0)
      { S7_Templates := "SrcType := Time" } GT_Contact(in1 := "AI_HMI_SP_Time_Khuay_Bon3", in2 := T#0s)
      { S7_Templates := "SrcType := Time" } GT_Contact(in1 := "AI_HMI_SP_Time_Fwd", in2 := T#0s)
      { S7_Templates := "SrcType := Time" } GT_Contact(in1 := "AI_HMI_SP_Time_Rev", in2 := T#0s)
      { S7_Templates := "SrcType := Time" } GT_Contact(in1 := "AI_HMI_SP_Time_Sterilize", in2 := T#0s)
      Coil( "AI_PLC2_SP_Valid" )
   END_RUNG
   // the same network as SCL:
   "AI_PLC2_SP_Valid" := ("AI_HMI_SP_PLC2_Nuoc_Bon3" > 0.0) AND ("AI_HMI_SP_PLC2_Nuoc_Bon4" > 0.0) AND ("AI_HMI_SP_PLC2_Toc_Do_Bon3" > 0.0) AND ("AI_HMI_SP_PLC2_Toc_Do_Bon4_Main" > 0.0) AND ("AI_HMI_SP_PLC2_Nhiet_Do_Bon4" > 0.0) AND ("AI_HMI_SP_Time_Khuay_Bon3" > T#0s) AND ("AI_HMI_SP_Time_Fwd" > T#0s) AND ("AI_HMI_SP_Time_Rev" > T#0s) AND ("AI_HMI_SP_Time_Sterilize" > T#0s);
END_REGION

REGION Network 46: Nhận cạnh lên nút nhấn Start PLC2
   RUNG wire#powerrail
      Contact( "AI_Nut_Khoi_Dong_Nhan_Eff" )
      P_Trig( "AI_PLC2_Start_Edge_Old" )
      Coil( "AI_PLC2_Start_Edge_Edge" )
   END_RUNG
   // the same network as SCL:
   #_w1 := "AI_Nut_Khoi_Dong_Nhan_Eff" AND NOT "AI_PLC2_Start_Edge_Old";   // rising edge
   "AI_PLC2_Start_Edge_Old" := "AI_Nut_Khoi_Dong_Nhan_Eff";
   "AI_PLC2_Start_Edge_Edge" := #_w1;
END_REGION

REGION Network 47: Khởi động chu trình PLC2 - Set Auto Enable
   RUNG wire#powerrail
      { S7_Templates := "SrcType := Int" } EQ_Contact(in1 := "AI_PLC2_State", in2 := 0)
      Contact( "AI_PLC2_Start_Edge_Edge" )
      I_Contact( "AI_PLC2_Loi_Tong" )
      Contact( "AI_PLC2_SP_Valid" )
      S_Coil( "AI_PLC2_Auto_Enable" )
   END_RUNG
   // the same network as SCL:
   IF ("AI_PLC2_State" = 0) AND "AI_PLC2_Start_Edge_Edge" AND NOT "AI_PLC2_Loi_Tong" AND "AI_PLC2_SP_Valid" THEN
       "AI_PLC2_Auto_Enable" := TRUE;
   END_IF;
END_REGION

REGION Network 48: Khởi động chu trình PLC2 - Chuyển sang State 10
   RUNG wire#powerrail
      { S7_Templates := "SrcType := Int" } EQ_Contact(in1 := "AI_PLC2_State", in2 := 0)
      Contact( "AI_PLC2_Start_Edge_Edge" )
      I_Contact( "AI_PLC2_Loi_Tong" )
      Contact( "AI_PLC2_SP_Valid" )
      { S7_GenerateENO := "TRUE" } Move(in := 10, out1 => "AI_PLC2_State")
   END_RUNG
   // the same network as SCL:
   IF ("AI_PLC2_State" = 0) AND "AI_PLC2_Start_Edge_Edge" AND NOT "AI_PLC2_Loi_Tong" AND "AI_PLC2_SP_Valid" THEN
       "AI_PLC2_State" := 10;
   END_IF;
END_REGION

REGION Network 49: Báo lỗi setpoint PLC2 khi bấm Start
   RUNG wire#powerrail
      Contact( "AI_PLC2_Start_Edge_Edge" )
      I_Contact( "AI_PLC2_Loi_Tong" )
      I_Contact( "AI_PLC2_SP_Valid" )
      S_Coil( "AI_PLC2_Loi_Setpoint" )
   END_RUNG
   // the same network as SCL:
   IF "AI_PLC2_Start_Edge_Edge" AND NOT "AI_PLC2_Loi_Tong" AND NOT "AI_PLC2_SP_Valid" THEN
       "AI_PLC2_Loi_Setpoint" := TRUE;
   END_IF;
END_REGION

REGION Network 50: Stop PLC2 từ HMI dùng chung
   RUNG wire#powerrail
      Contact( "AI_Nut_Dung_Nhan_Eff" )
      { S7_GenerateENO := "TRUE" } Move(in := 0, out1 => "AI_PLC2_State")
   END_RUNG
   // the same network as SCL:
   IF "AI_Nut_Dung_Nhan_Eff" THEN "AI_PLC2_State" := 0; END_IF;
END_REGION

REGION Network 51: Stop PLC2 - reset Auto Enable
   RUNG wire#powerrail
      Contact( "AI_Nut_Dung_Nhan_Eff" )
      R_Coil( "AI_PLC2_Auto_Enable" )
   END_RUNG
   // the same network as SCL:
   IF "AI_Nut_Dung_Nhan_Eff" THEN "AI_PLC2_Auto_Enable" := FALSE; END_IF;
END_REGION

REGION Network 52: Tạo tín hiệu Stop active PLC2
   RUNG wire#powerrail
      Contact( "AI_Nut_Dung_Nhan_Eff" )
      Coil( "AI_PLC2_Stop_Active" )
   END_RUNG
   // the same network as SCL:
   "AI_PLC2_Stop_Active" := "AI_Nut_Dung_Nhan_Eff";
END_REGION

REGION Network 53: Stop PLC2 - reset AI_V3240_Nuoc_Bon3
   RUNG wire#powerrail
      Contact( "AI_PLC2_Stop_Active" )
      R_Coil( "AI_V3240_Nuoc_Bon3" )
   END_RUNG
   // the same network as SCL:
   IF "AI_PLC2_Stop_Active" THEN "AI_V3240_Nuoc_Bon3" := FALSE; END_IF;
END_REGION

REGION Network 54: Stop PLC2 - reset AI_V3242_Xa_Bon3
   RUNG wire#powerrail
      Contact( "AI_PLC2_Stop_Active" )
      R_Coil( "AI_V3242_Xa_Bon3" )
   END_RUNG
   // the same network as SCL:
   IF "AI_PLC2_Stop_Active" THEN "AI_V3242_Xa_Bon3" := FALSE; END_IF;
END_REGION

REGION Network 55: Stop PLC2 - reset AI_V3243_Xa_Bon3
   RUNG wire#powerrail
      Contact( "AI_PLC2_Stop_Active" )
      R_Coil( "AI_V3243_Xa_Bon3" )
   END_RUNG
   // the same network as SCL:
   IF "AI_PLC2_Stop_Active" THEN "AI_V3243_Xa_Bon3" := FALSE; END_IF;
END_REGION

REGION Network 56: Stop PLC2 - reset AI_V3244_Xa_Bon3
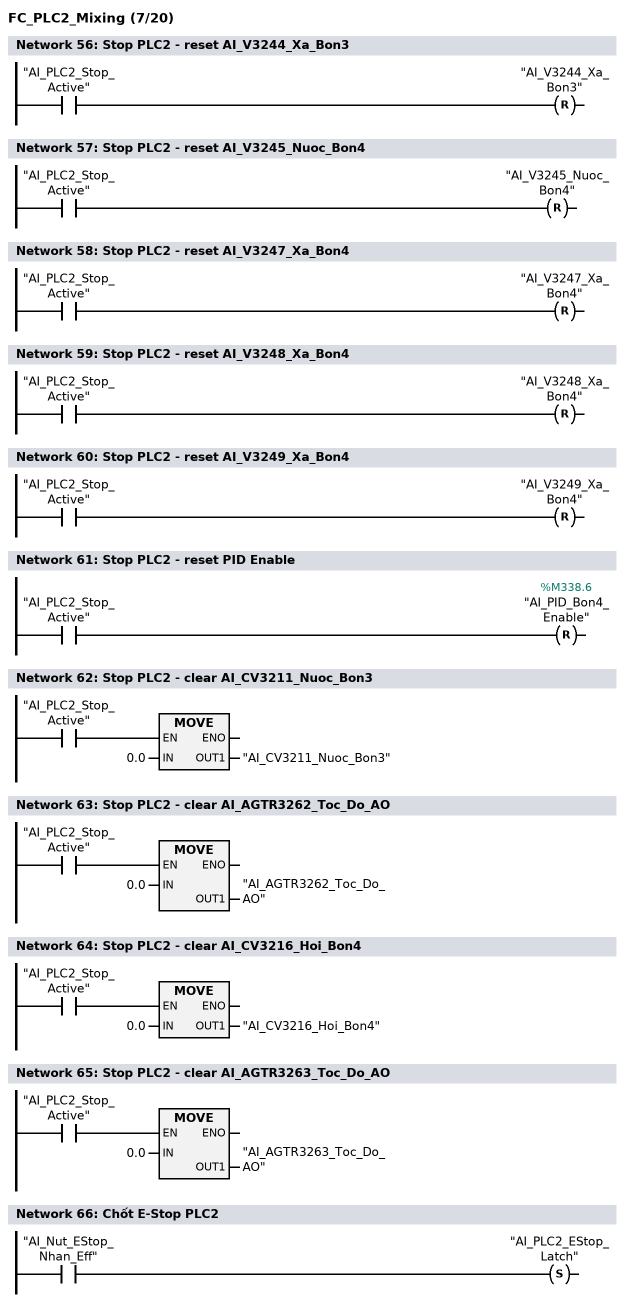
   RUNG wire#powerrail
      Contact( "AI_PLC2_Stop_Active" )
      R_Coil( "AI_V3244_Xa_Bon3" )
   END_RUNG
   // the same network as SCL:
   IF "AI_PLC2_Stop_Active" THEN "AI_V3244_Xa_Bon3" := FALSE; END_IF;
END_REGION

REGION Network 57: Stop PLC2 - reset AI_V3245_Nuoc_Bon4
   RUNG wire#powerrail
      Contact( "AI_PLC2_Stop_Active" )
      R_Coil( "AI_V3245_Nuoc_Bon4" )
   END_RUNG
   // the same network as SCL:
   IF "AI_PLC2_Stop_Active" THEN "AI_V3245_Nuoc_Bon4" := FALSE; END_IF;
END_REGION

REGION Network 58: Stop PLC2 - reset AI_V3247_Xa_Bon4
   RUNG wire#powerrail
      Contact( "AI_PLC2_Stop_Active" )
      R_Coil( "AI_V3247_Xa_Bon4" )
   END_RUNG
   // the same network as SCL:
   IF "AI_PLC2_Stop_Active" THEN "AI_V3247_Xa_Bon4" := FALSE; END_IF;
END_REGION

REGION Network 59: Stop PLC2 - reset AI_V3248_Xa_Bon4
   RUNG wire#powerrail
      Contact( "AI_PLC2_Stop_Active" )
      R_Coil( "AI_V3248_Xa_Bon4" )
   END_RUNG
   // the same network as SCL:
   IF "AI_PLC2_Stop_Active" THEN "AI_V3248_Xa_Bon4" := FALSE; END_IF;
END_REGION

REGION Network 60: Stop PLC2 - reset AI_V3249_Xa_Bon4
   RUNG wire#powerrail
      Contact( "AI_PLC2_Stop_Active" )
      R_Coil( "AI_V3249_Xa_Bon4" )
   END_RUNG
   // the same network as SCL:
   IF "AI_PLC2_Stop_Active" THEN "AI_V3249_Xa_Bon4" := FALSE; END_IF;
END_REGION

REGION Network 61: Stop PLC2 - reset PID Enable
   RUNG wire#powerrail
      Contact( "AI_PLC2_Stop_Active" )
      R_Coil( "AI_PID_Bon4_Enable" )
   END_RUNG
   // the same network as SCL:
   IF "AI_PLC2_Stop_Active" THEN "AI_PID_Bon4_Enable" := FALSE; END_IF;
END_REGION

REGION Network 62: Stop PLC2 - clear AI_CV3211_Nuoc_Bon3
   RUNG wire#powerrail
      Contact( "AI_PLC2_Stop_Active" )
      { S7_GenerateENO := "TRUE" } Move(in := 0.0, out1 => "AI_CV3211_Nuoc_Bon3")
   END_RUNG
   // the same network as SCL:
   IF "AI_PLC2_Stop_Active" THEN "AI_CV3211_Nuoc_Bon3" := 0.0; END_IF;
END_REGION

REGION Network 63: Stop PLC2 - clear AI_AGTR3262_Toc_Do_AO
   RUNG wire#powerrail
      Contact( "AI_PLC2_Stop_Active" )
      { S7_GenerateENO := "TRUE" } Move(in := 0.0, out1 => "AI_AGTR3262_Toc_Do_AO")
   END_RUNG
   // the same network as SCL:
   IF "AI_PLC2_Stop_Active" THEN "AI_AGTR3262_Toc_Do_AO" := 0.0; END_IF;
END_REGION

REGION Network 64: Stop PLC2 - clear AI_CV3216_Hoi_Bon4
   RUNG wire#powerrail
      Contact( "AI_PLC2_Stop_Active" )
      { S7_GenerateENO := "TRUE" } Move(in := 0.0, out1 => "AI_CV3216_Hoi_Bon4")
   END_RUNG
   // the same network as SCL:
   IF "AI_PLC2_Stop_Active" THEN "AI_CV3216_Hoi_Bon4" := 0.0; END_IF;
END_REGION

REGION Network 65: Stop PLC2 - clear AI_AGTR3263_Toc_Do_AO
   RUNG wire#powerrail
      Contact( "AI_PLC2_Stop_Active" )
      { S7_GenerateENO := "TRUE" } Move(in := 0.0, out1 => "AI_AGTR3263_Toc_Do_AO")
   END_RUNG
   // the same network as SCL:
   IF "AI_PLC2_Stop_Active" THEN "AI_AGTR3263_Toc_Do_AO" := 0.0; END_IF;
END_REGION

REGION Network 66: Chốt E-Stop PLC2
   RUNG wire#powerrail
      Contact( "AI_Nut_EStop_Nhan_Eff" )
      S_Coil( "AI_PLC2_EStop_Latch" )
   END_RUNG
   // the same network as SCL:
   IF "AI_Nut_EStop_Nhan_Eff" THEN "AI_PLC2_EStop_Latch" := TRUE; END_IF;
END_REGION

REGION Network 67: Reset chốt E-Stop PLC2 an toàn (Vật lý)
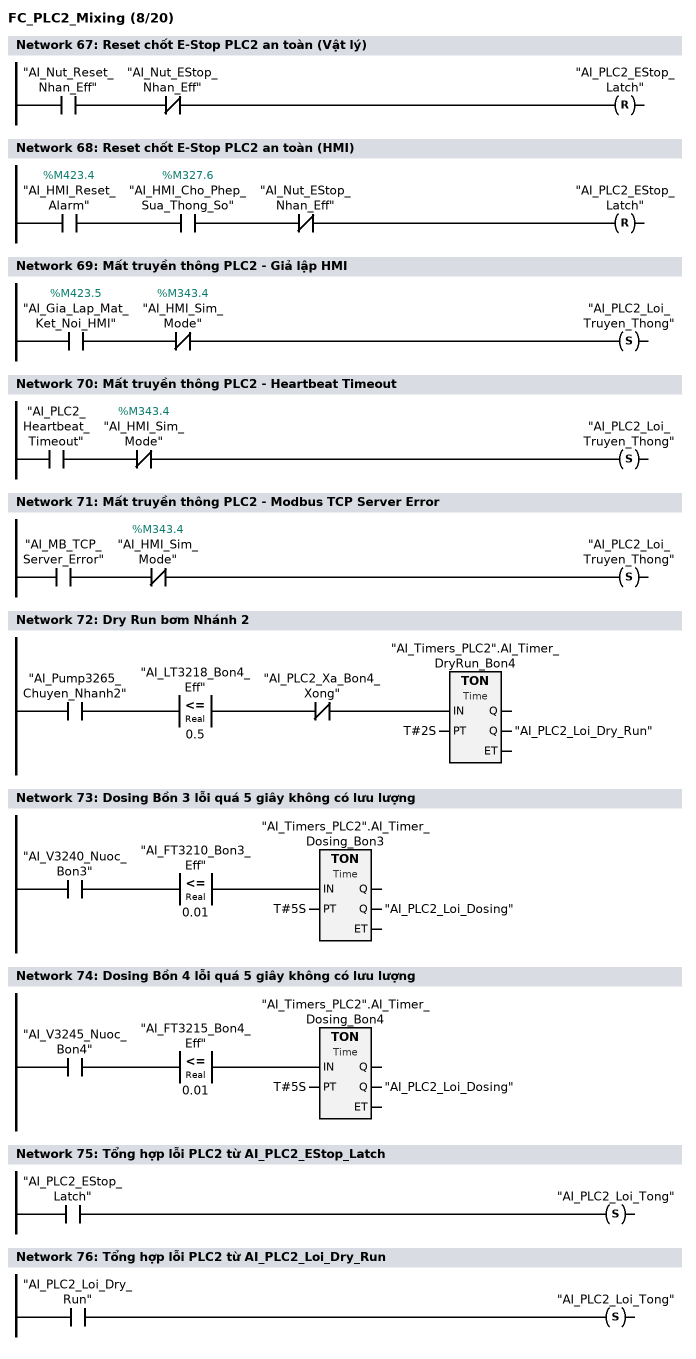
   RUNG wire#powerrail
      Contact( "AI_Nut_Reset_Nhan_Eff" )
      I_Contact( "AI_Nut_EStop_Nhan_Eff" )
      R_Coil( "AI_PLC2_EStop_Latch" )
   END_RUNG
   // the same network as SCL:
   IF "AI_Nut_Reset_Nhan_Eff" AND NOT "AI_Nut_EStop_Nhan_Eff" THEN "AI_PLC2_EStop_Latch" := FALSE; END_IF;
END_REGION

REGION Network 68: Reset chốt E-Stop PLC2 an toàn (HMI)
   RUNG wire#powerrail
      Contact( "AI_HMI_Reset_Alarm" )
      Contact( "AI_HMI_Cho_Phep_Sua_Thong_So" )
      I_Contact( "AI_Nut_EStop_Nhan_Eff" )
      R_Coil( "AI_PLC2_EStop_Latch" )
   END_RUNG
   // the same network as SCL:
   IF "AI_HMI_Reset_Alarm" AND "AI_HMI_Cho_Phep_Sua_Thong_So" AND NOT "AI_Nut_EStop_Nhan_Eff" THEN
       "AI_PLC2_EStop_Latch" := FALSE;
   END_IF;
END_REGION

REGION Network 69: Mất truyền thông PLC2 - Giả lập HMI
   RUNG wire#powerrail
      Contact( "AI_Gia_Lap_Mat_Ket_Noi_HMI" )
      I_Contact( "AI_HMI_Sim_Mode" )
      S_Coil( "AI_PLC2_Loi_Truyen_Thong" )
   END_RUNG
   // the same network as SCL:
   IF "AI_Gia_Lap_Mat_Ket_Noi_HMI" AND NOT "AI_HMI_Sim_Mode" THEN "AI_PLC2_Loi_Truyen_Thong" := TRUE; END_IF;
END_REGION

REGION Network 70: Mất truyền thông PLC2 - Heartbeat Timeout
   RUNG wire#powerrail
      Contact( "AI_PLC2_Heartbeat_Timeout" )
      I_Contact( "AI_HMI_Sim_Mode" )
      S_Coil( "AI_PLC2_Loi_Truyen_Thong" )
   END_RUNG
   // the same network as SCL:
   IF "AI_PLC2_Heartbeat_Timeout" AND NOT "AI_HMI_Sim_Mode" THEN "AI_PLC2_Loi_Truyen_Thong" := TRUE; END_IF;
END_REGION

REGION Network 71: Mất truyền thông PLC2 - Modbus TCP Server Error
   RUNG wire#powerrail
      Contact( "AI_MB_TCP_Server_Error" )
      I_Contact( "AI_HMI_Sim_Mode" )
      S_Coil( "AI_PLC2_Loi_Truyen_Thong" )
   END_RUNG
   // the same network as SCL:
   IF "AI_MB_TCP_Server_Error" AND NOT "AI_HMI_Sim_Mode" THEN "AI_PLC2_Loi_Truyen_Thong" := TRUE; END_IF;
END_REGION

REGION Network 72: Dry Run bơm Nhánh 2
   RUNG wire#powerrail
      Contact( "AI_Pump3265_Chuyen_Nhanh2" )
      { S7_Templates := "SrcType := Real" } LE_Contact(in1 := "AI_LT3218_Bon4_Eff", in2 := 0.5)
      I_Contact( "AI_PLC2_Xa_Bon4_Xong" )
      { S7_Templates := "time_type := Time" } "AI_Timers_PLC2".AI_Timer_DryRun_Bon4.TON(pt := T#2S, q => "AI_PLC2_Loi_Dry_Run", et =>)
   END_RUNG
   // the same network as SCL:
   "AI_Timers_PLC2".AI_Timer_DryRun_Bon4.TON(IN := "AI_Pump3265_Chuyen_Nhanh2" AND ("AI_LT3218_Bon4_Eff" <= 0.5) AND NOT "AI_PLC2_Xa_Bon4_Xong",
                           PT := T#2S,
                           Q => "AI_PLC2_Loi_Dry_Run");
END_REGION

REGION Network 73: Dosing Bồn 3 lỗi quá 5 giây không có lưu lượng
   RUNG wire#powerrail
      Contact( "AI_V3240_Nuoc_Bon3" )
      { S7_Templates := "SrcType := Real" } LE_Contact(in1 := "AI_FT3210_Bon3_Eff", in2 := 0.01)
      { S7_Templates := "time_type := Time" } "AI_Timers_PLC2".AI_Timer_Dosing_Bon3.TON(pt := T#5S, q => "AI_PLC2_Loi_Dosing", et =>)
   END_RUNG
   // the same network as SCL:
   "AI_Timers_PLC2".AI_Timer_Dosing_Bon3.TON(IN := "AI_V3240_Nuoc_Bon3" AND ("AI_FT3210_Bon3_Eff" <= 0.01),
                           PT := T#5S,
                           Q => "AI_PLC2_Loi_Dosing");
END_REGION

REGION Network 74: Dosing Bồn 4 lỗi quá 5 giây không có lưu lượng
   RUNG wire#powerrail
      Contact( "AI_V3245_Nuoc_Bon4" )
      { S7_Templates := "SrcType := Real" } LE_Contact(in1 := "AI_FT3215_Bon4_Eff", in2 := 0.01)
      { S7_Templates := "time_type := Time" } "AI_Timers_PLC2".AI_Timer_Dosing_Bon4.TON(pt := T#5S, q => "AI_PLC2_Loi_Dosing", et =>)
   END_RUNG
   // the same network as SCL:
   "AI_Timers_PLC2".AI_Timer_Dosing_Bon4.TON(IN := "AI_V3245_Nuoc_Bon4" AND ("AI_FT3215_Bon4_Eff" <= 0.01),
                           PT := T#5S,
                           Q => "AI_PLC2_Loi_Dosing");
END_REGION

REGION Network 75: Tổng hợp lỗi PLC2 từ AI_PLC2_EStop_Latch
   RUNG wire#powerrail
      Contact( "AI_PLC2_EStop_Latch" )
      S_Coil( "AI_PLC2_Loi_Tong" )
   END_RUNG
   // the same network as SCL:
   IF "AI_PLC2_EStop_Latch" THEN "AI_PLC2_Loi_Tong" := TRUE; END_IF;
END_REGION

REGION Network 76: Tổng hợp lỗi PLC2 từ AI_PLC2_Loi_Dry_Run
   RUNG wire#powerrail
      Contact( "AI_PLC2_Loi_Dry_Run" )
      S_Coil( "AI_PLC2_Loi_Tong" )
   END_RUNG
   // the same network as SCL:
   IF "AI_PLC2_Loi_Dry_Run" THEN "AI_PLC2_Loi_Tong" := TRUE; END_IF;
END_REGION

REGION Network 77: Tổng hợp lỗi PLC2 từ AI_PLC2_Loi_Dosing
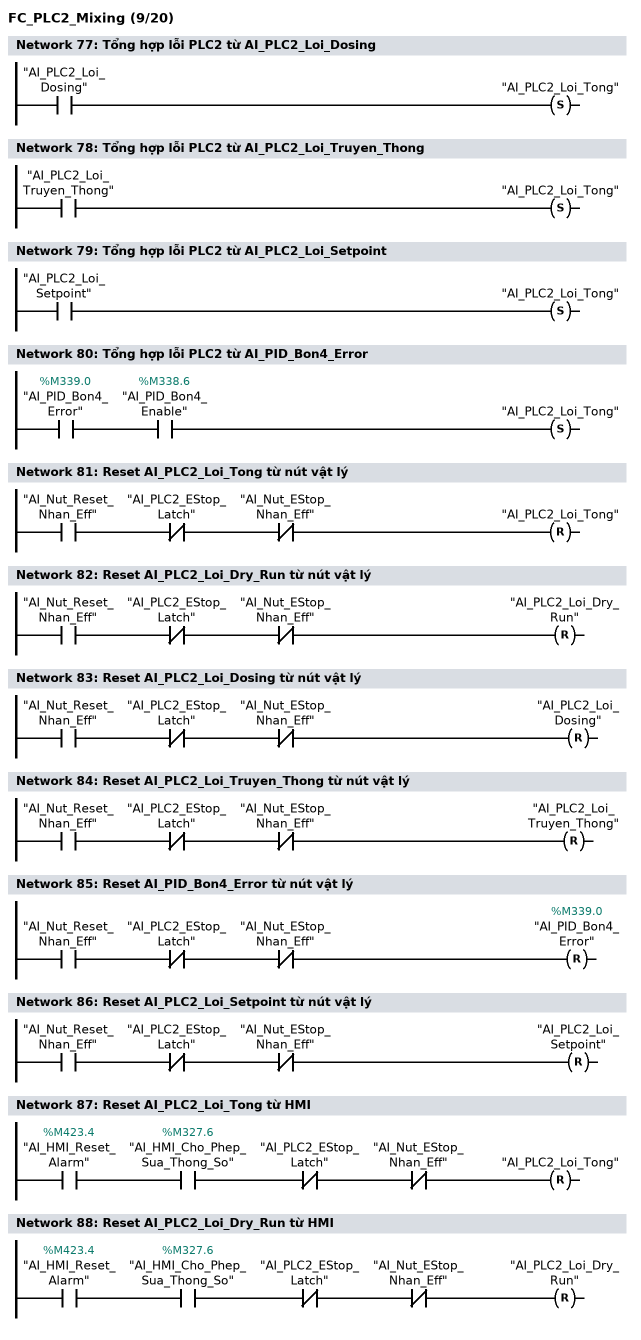
   RUNG wire#powerrail
      Contact( "AI_PLC2_Loi_Dosing" )
      S_Coil( "AI_PLC2_Loi_Tong" )
   END_RUNG
   // the same network as SCL:
   IF "AI_PLC2_Loi_Dosing" THEN "AI_PLC2_Loi_Tong" := TRUE; END_IF;
END_REGION

REGION Network 78: Tổng hợp lỗi PLC2 từ AI_PLC2_Loi_Truyen_Thong
   RUNG wire#powerrail
      Contact( "AI_PLC2_Loi_Truyen_Thong" )
      S_Coil( "AI_PLC2_Loi_Tong" )
   END_RUNG
   // the same network as SCL:
   IF "AI_PLC2_Loi_Truyen_Thong" THEN "AI_PLC2_Loi_Tong" := TRUE; END_IF;
END_REGION

REGION Network 79: Tổng hợp lỗi PLC2 từ AI_PLC2_Loi_Setpoint
   RUNG wire#powerrail
      Contact( "AI_PLC2_Loi_Setpoint" )
      S_Coil( "AI_PLC2_Loi_Tong" )
   END_RUNG
   // the same network as SCL:
   IF "AI_PLC2_Loi_Setpoint" THEN "AI_PLC2_Loi_Tong" := TRUE; END_IF;
END_REGION

REGION Network 80: Tổng hợp lỗi PLC2 từ AI_PID_Bon4_Error
   RUNG wire#powerrail
      Contact( "AI_PID_Bon4_Error" )
      Contact( "AI_PID_Bon4_Enable" )
      S_Coil( "AI_PLC2_Loi_Tong" )
   END_RUNG
   // the same network as SCL:
   IF "AI_PID_Bon4_Error" AND "AI_PID_Bon4_Enable" THEN "AI_PLC2_Loi_Tong" := TRUE; END_IF;
END_REGION

REGION Network 81: Reset AI_PLC2_Loi_Tong từ nút vật lý
   RUNG wire#powerrail
      Contact( "AI_Nut_Reset_Nhan_Eff" )
      I_Contact( "AI_PLC2_EStop_Latch" )
      I_Contact( "AI_Nut_EStop_Nhan_Eff" )
      R_Coil( "AI_PLC2_Loi_Tong" )
   END_RUNG
   // the same network as SCL:
   IF "AI_Nut_Reset_Nhan_Eff" AND NOT "AI_PLC2_EStop_Latch" AND NOT "AI_Nut_EStop_Nhan_Eff" THEN
       "AI_PLC2_Loi_Tong" := FALSE;
   END_IF;
END_REGION

REGION Network 82: Reset AI_PLC2_Loi_Dry_Run từ nút vật lý
   RUNG wire#powerrail
      Contact( "AI_Nut_Reset_Nhan_Eff" )
      I_Contact( "AI_PLC2_EStop_Latch" )
      I_Contact( "AI_Nut_EStop_Nhan_Eff" )
      R_Coil( "AI_PLC2_Loi_Dry_Run" )
   END_RUNG
   // the same network as SCL:
   IF "AI_Nut_Reset_Nhan_Eff" AND NOT "AI_PLC2_EStop_Latch" AND NOT "AI_Nut_EStop_Nhan_Eff" THEN
       "AI_PLC2_Loi_Dry_Run" := FALSE;
   END_IF;
END_REGION

REGION Network 83: Reset AI_PLC2_Loi_Dosing từ nút vật lý
   RUNG wire#powerrail
      Contact( "AI_Nut_Reset_Nhan_Eff" )
      I_Contact( "AI_PLC2_EStop_Latch" )
      I_Contact( "AI_Nut_EStop_Nhan_Eff" )
      R_Coil( "AI_PLC2_Loi_Dosing" )
   END_RUNG
   // the same network as SCL:
   IF "AI_Nut_Reset_Nhan_Eff" AND NOT "AI_PLC2_EStop_Latch" AND NOT "AI_Nut_EStop_Nhan_Eff" THEN
       "AI_PLC2_Loi_Dosing" := FALSE;
   END_IF;
END_REGION

REGION Network 84: Reset AI_PLC2_Loi_Truyen_Thong từ nút vật lý
   RUNG wire#powerrail
      Contact( "AI_Nut_Reset_Nhan_Eff" )
      I_Contact( "AI_PLC2_EStop_Latch" )
      I_Contact( "AI_Nut_EStop_Nhan_Eff" )
      R_Coil( "AI_PLC2_Loi_Truyen_Thong" )
   END_RUNG
   // the same network as SCL:
   IF "AI_Nut_Reset_Nhan_Eff" AND NOT "AI_PLC2_EStop_Latch" AND NOT "AI_Nut_EStop_Nhan_Eff" THEN
       "AI_PLC2_Loi_Truyen_Thong" := FALSE;
   END_IF;
END_REGION

REGION Network 85: Reset AI_PID_Bon4_Error từ nút vật lý
   RUNG wire#powerrail
      Contact( "AI_Nut_Reset_Nhan_Eff" )
      I_Contact( "AI_PLC2_EStop_Latch" )
      I_Contact( "AI_Nut_EStop_Nhan_Eff" )
      R_Coil( "AI_PID_Bon4_Error" )
   END_RUNG
   // the same network as SCL:
   IF "AI_Nut_Reset_Nhan_Eff" AND NOT "AI_PLC2_EStop_Latch" AND NOT "AI_Nut_EStop_Nhan_Eff" THEN
       "AI_PID_Bon4_Error" := FALSE;
   END_IF;
END_REGION

REGION Network 86: Reset AI_PLC2_Loi_Setpoint từ nút vật lý
   RUNG wire#powerrail
      Contact( "AI_Nut_Reset_Nhan_Eff" )
      I_Contact( "AI_PLC2_EStop_Latch" )
      I_Contact( "AI_Nut_EStop_Nhan_Eff" )
      R_Coil( "AI_PLC2_Loi_Setpoint" )
   END_RUNG
   // the same network as SCL:
   IF "AI_Nut_Reset_Nhan_Eff" AND NOT "AI_PLC2_EStop_Latch" AND NOT "AI_Nut_EStop_Nhan_Eff" THEN
       "AI_PLC2_Loi_Setpoint" := FALSE;
   END_IF;
END_REGION

REGION Network 87: Reset AI_PLC2_Loi_Tong từ HMI
   RUNG wire#powerrail
      Contact( "AI_HMI_Reset_Alarm" )
      Contact( "AI_HMI_Cho_Phep_Sua_Thong_So" )
      I_Contact( "AI_PLC2_EStop_Latch" )
      I_Contact( "AI_Nut_EStop_Nhan_Eff" )
      R_Coil( "AI_PLC2_Loi_Tong" )
   END_RUNG
   // the same network as SCL:
   IF "AI_HMI_Reset_Alarm" AND "AI_HMI_Cho_Phep_Sua_Thong_So" AND NOT "AI_PLC2_EStop_Latch" AND NOT "AI_Nut_EStop_Nhan_Eff" THEN
       "AI_PLC2_Loi_Tong" := FALSE;
   END_IF;
END_REGION

REGION Network 88: Reset AI_PLC2_Loi_Dry_Run từ HMI
   RUNG wire#powerrail
      Contact( "AI_HMI_Reset_Alarm" )
      Contact( "AI_HMI_Cho_Phep_Sua_Thong_So" )
      I_Contact( "AI_PLC2_EStop_Latch" )
      I_Contact( "AI_Nut_EStop_Nhan_Eff" )
      R_Coil( "AI_PLC2_Loi_Dry_Run" )
   END_RUNG
   // the same network as SCL:
   IF "AI_HMI_Reset_Alarm" AND "AI_HMI_Cho_Phep_Sua_Thong_So" AND NOT "AI_PLC2_EStop_Latch" AND NOT "AI_Nut_EStop_Nhan_Eff" THEN
       "AI_PLC2_Loi_Dry_Run" := FALSE;
   END_IF;
END_REGION

REGION Network 89: Reset AI_PLC2_Loi_Dosing từ HMI
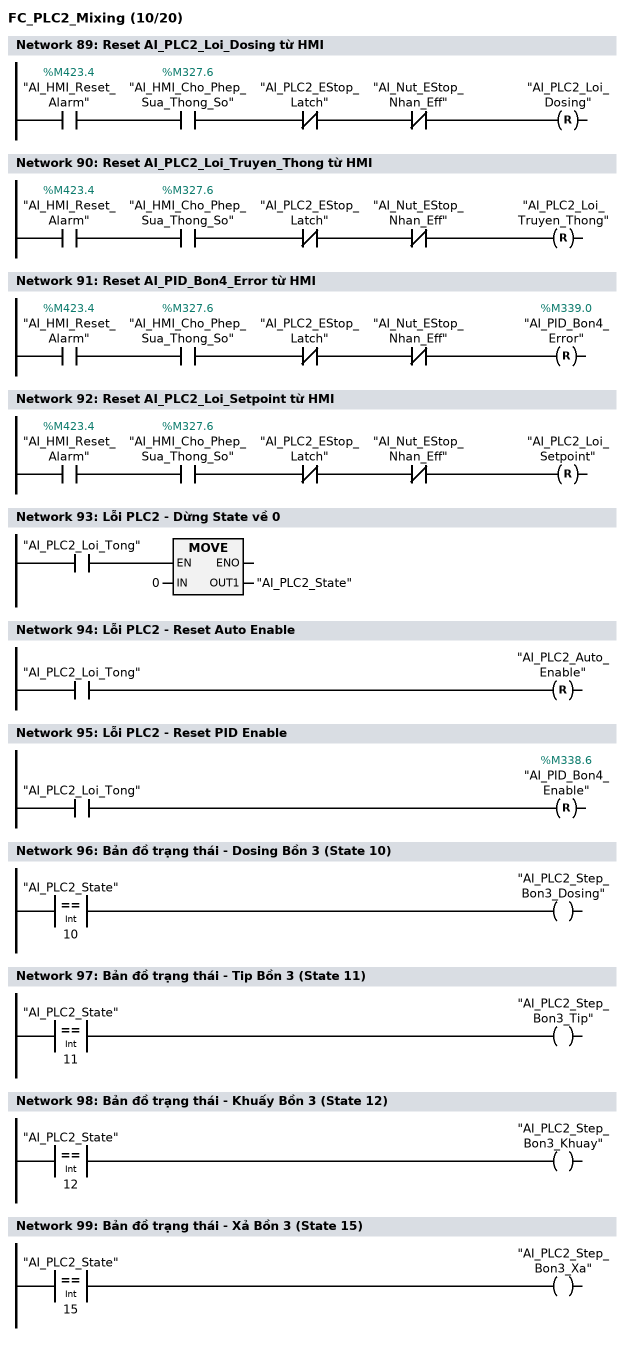
   RUNG wire#powerrail
      Contact( "AI_HMI_Reset_Alarm" )
      Contact( "AI_HMI_Cho_Phep_Sua_Thong_So" )
      I_Contact( "AI_PLC2_EStop_Latch" )
      I_Contact( "AI_Nut_EStop_Nhan_Eff" )
      R_Coil( "AI_PLC2_Loi_Dosing" )
   END_RUNG
   // the same network as SCL:
   IF "AI_HMI_Reset_Alarm" AND "AI_HMI_Cho_Phep_Sua_Thong_So" AND NOT "AI_PLC2_EStop_Latch" AND NOT "AI_Nut_EStop_Nhan_Eff" THEN
       "AI_PLC2_Loi_Dosing" := FALSE;
   END_IF;
END_REGION

REGION Network 90: Reset AI_PLC2_Loi_Truyen_Thong từ HMI
   RUNG wire#powerrail
      Contact( "AI_HMI_Reset_Alarm" )
      Contact( "AI_HMI_Cho_Phep_Sua_Thong_So" )
      I_Contact( "AI_PLC2_EStop_Latch" )
      I_Contact( "AI_Nut_EStop_Nhan_Eff" )
      R_Coil( "AI_PLC2_Loi_Truyen_Thong" )
   END_RUNG
   // the same network as SCL:
   IF "AI_HMI_Reset_Alarm" AND "AI_HMI_Cho_Phep_Sua_Thong_So" AND NOT "AI_PLC2_EStop_Latch" AND NOT "AI_Nut_EStop_Nhan_Eff" THEN
       "AI_PLC2_Loi_Truyen_Thong" := FALSE;
   END_IF;
END_REGION

REGION Network 91: Reset AI_PID_Bon4_Error từ HMI
   RUNG wire#powerrail
      Contact( "AI_HMI_Reset_Alarm" )
      Contact( "AI_HMI_Cho_Phep_Sua_Thong_So" )
      I_Contact( "AI_PLC2_EStop_Latch" )
      I_Contact( "AI_Nut_EStop_Nhan_Eff" )
      R_Coil( "AI_PID_Bon4_Error" )
   END_RUNG
   // the same network as SCL:
   IF "AI_HMI_Reset_Alarm" AND "AI_HMI_Cho_Phep_Sua_Thong_So" AND NOT "AI_PLC2_EStop_Latch" AND NOT "AI_Nut_EStop_Nhan_Eff" THEN
       "AI_PID_Bon4_Error" := FALSE;
   END_IF;
END_REGION

REGION Network 92: Reset AI_PLC2_Loi_Setpoint từ HMI
   RUNG wire#powerrail
      Contact( "AI_HMI_Reset_Alarm" )
      Contact( "AI_HMI_Cho_Phep_Sua_Thong_So" )
      I_Contact( "AI_PLC2_EStop_Latch" )
      I_Contact( "AI_Nut_EStop_Nhan_Eff" )
      R_Coil( "AI_PLC2_Loi_Setpoint" )
   END_RUNG
   // the same network as SCL:
   IF "AI_HMI_Reset_Alarm" AND "AI_HMI_Cho_Phep_Sua_Thong_So" AND NOT "AI_PLC2_EStop_Latch" AND NOT "AI_Nut_EStop_Nhan_Eff" THEN
       "AI_PLC2_Loi_Setpoint" := FALSE;
   END_IF;
END_REGION

REGION Network 93: Lỗi PLC2 - Dừng State về 0
   RUNG wire#powerrail
      Contact( "AI_PLC2_Loi_Tong" )
      { S7_GenerateENO := "TRUE" } Move(in := 0, out1 => "AI_PLC2_State")
   END_RUNG
   // the same network as SCL:
   IF "AI_PLC2_Loi_Tong" THEN "AI_PLC2_State" := 0; END_IF;
END_REGION

REGION Network 94: Lỗi PLC2 - Reset Auto Enable
   RUNG wire#powerrail
      Contact( "AI_PLC2_Loi_Tong" )
      R_Coil( "AI_PLC2_Auto_Enable" )
   END_RUNG
   // the same network as SCL:
   IF "AI_PLC2_Loi_Tong" THEN "AI_PLC2_Auto_Enable" := FALSE; END_IF;
END_REGION

REGION Network 95: Lỗi PLC2 - Reset PID Enable
   RUNG wire#powerrail
      Contact( "AI_PLC2_Loi_Tong" )
      R_Coil( "AI_PID_Bon4_Enable" )
   END_RUNG
   // the same network as SCL:
   IF "AI_PLC2_Loi_Tong" THEN "AI_PID_Bon4_Enable" := FALSE; END_IF;
END_REGION

REGION Network 96: Bản đồ trạng thái - Dosing Bồn 3 (State 10)
   RUNG wire#powerrail
      { S7_Templates := "SrcType := Int" } EQ_Contact(in1 := "AI_PLC2_State", in2 := 10)
      Coil( "AI_PLC2_Step_Bon3_Dosing" )
   END_RUNG
   // the same network as SCL:
   "AI_PLC2_Step_Bon3_Dosing" := "AI_PLC2_State" = 10;
END_REGION

REGION Network 97: Bản đồ trạng thái - Tip Bồn 3 (State 11)
   RUNG wire#powerrail
      { S7_Templates := "SrcType := Int" } EQ_Contact(in1 := "AI_PLC2_State", in2 := 11)
      Coil( "AI_PLC2_Step_Bon3_Tip" )
   END_RUNG
   // the same network as SCL:
   "AI_PLC2_Step_Bon3_Tip" := "AI_PLC2_State" = 11;
END_REGION

REGION Network 98: Bản đồ trạng thái - Khuấy Bồn 3 (State 12)
   RUNG wire#powerrail
      { S7_Templates := "SrcType := Int" } EQ_Contact(in1 := "AI_PLC2_State", in2 := 12)
      Coil( "AI_PLC2_Step_Bon3_Khuay" )
   END_RUNG
   // the same network as SCL:
   "AI_PLC2_Step_Bon3_Khuay" := "AI_PLC2_State" = 12;
END_REGION

REGION Network 99: Bản đồ trạng thái - Xả Bồn 3 (State 15)
   RUNG wire#powerrail
      { S7_Templates := "SrcType := Int" } EQ_Contact(in1 := "AI_PLC2_State", in2 := 15)
      Coil( "AI_PLC2_Step_Bon3_Xa" )
   END_RUNG
   // the same network as SCL:
   "AI_PLC2_Step_Bon3_Xa" := "AI_PLC2_State" = 15;
END_REGION

REGION Network 100: Bản đồ trạng thái - Dosing Bồn 4 (State 20)
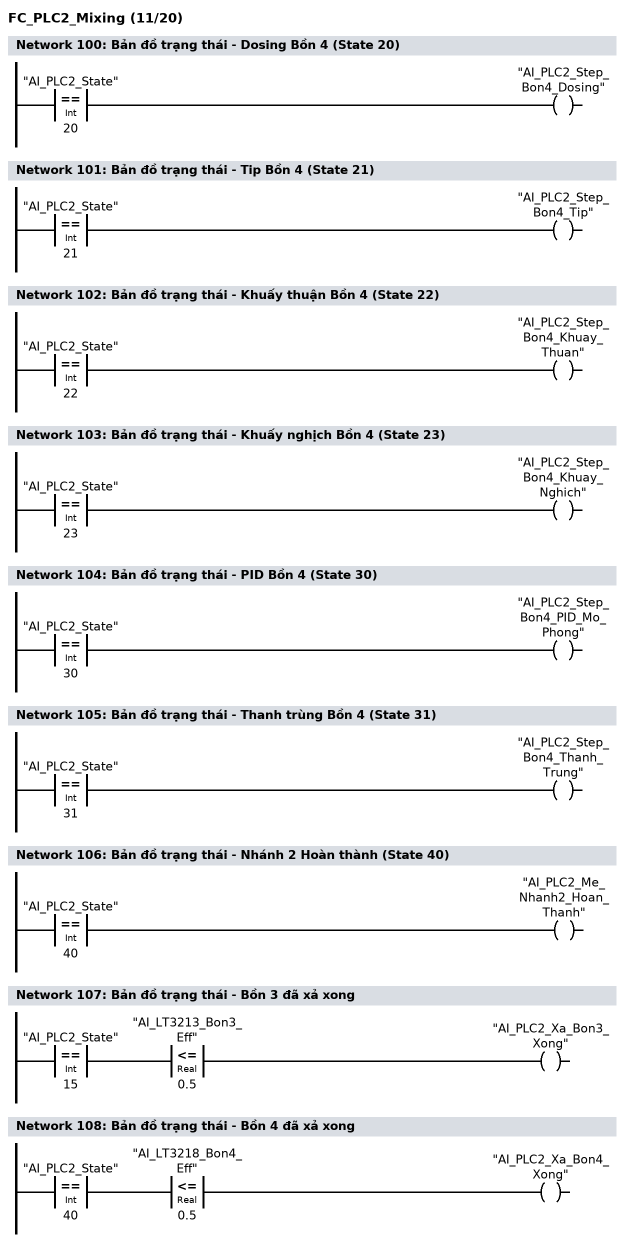
   RUNG wire#powerrail
      { S7_Templates := "SrcType := Int" } EQ_Contact(in1 := "AI_PLC2_State", in2 := 20)
      Coil( "AI_PLC2_Step_Bon4_Dosing" )
   END_RUNG
   // the same network as SCL:
   "AI_PLC2_Step_Bon4_Dosing" := "AI_PLC2_State" = 20;
END_REGION

REGION Network 101: Bản đồ trạng thái - Tip Bồn 4 (State 21)
   RUNG wire#powerrail
      { S7_Templates := "SrcType := Int" } EQ_Contact(in1 := "AI_PLC2_State", in2 := 21)
      Coil( "AI_PLC2_Step_Bon4_Tip" )
   END_RUNG
   // the same network as SCL:
   "AI_PLC2_Step_Bon4_Tip" := "AI_PLC2_State" = 21;
END_REGION

REGION Network 102: Bản đồ trạng thái - Khuấy thuận Bồn 4 (State 22)
   RUNG wire#powerrail
      { S7_Templates := "SrcType := Int" } EQ_Contact(in1 := "AI_PLC2_State", in2 := 22)
      Coil( "AI_PLC2_Step_Bon4_Khuay_Thuan" )
   END_RUNG
   // the same network as SCL:
   "AI_PLC2_Step_Bon4_Khuay_Thuan" := "AI_PLC2_State" = 22;
END_REGION

REGION Network 103: Bản đồ trạng thái - Khuấy nghịch Bồn 4 (State 23)
   RUNG wire#powerrail
      { S7_Templates := "SrcType := Int" } EQ_Contact(in1 := "AI_PLC2_State", in2 := 23)
      Coil( "AI_PLC2_Step_Bon4_Khuay_Nghich" )
   END_RUNG
   // the same network as SCL:
   "AI_PLC2_Step_Bon4_Khuay_Nghich" := "AI_PLC2_State" = 23;
END_REGION

REGION Network 104: Bản đồ trạng thái - PID Bồn 4 (State 30)
   RUNG wire#powerrail
      { S7_Templates := "SrcType := Int" } EQ_Contact(in1 := "AI_PLC2_State", in2 := 30)
      Coil( "AI_PLC2_Step_Bon4_PID_Mo_Phong" )
   END_RUNG
   // the same network as SCL:
   "AI_PLC2_Step_Bon4_PID_Mo_Phong" := "AI_PLC2_State" = 30;
END_REGION

REGION Network 105: Bản đồ trạng thái - Thanh trùng Bồn 4 (State 31)
   RUNG wire#powerrail
      { S7_Templates := "SrcType := Int" } EQ_Contact(in1 := "AI_PLC2_State", in2 := 31)
      Coil( "AI_PLC2_Step_Bon4_Thanh_Trung" )
   END_RUNG
   // the same network as SCL:
   "AI_PLC2_Step_Bon4_Thanh_Trung" := "AI_PLC2_State" = 31;
END_REGION

REGION Network 106: Bản đồ trạng thái - Nhánh 2 Hoàn thành (State 40)
   RUNG wire#powerrail
      { S7_Templates := "SrcType := Int" } EQ_Contact(in1 := "AI_PLC2_State", in2 := 40)
      Coil( "AI_PLC2_Me_Nhanh2_Hoan_Thanh" )
   END_RUNG
   // the same network as SCL:
   "AI_PLC2_Me_Nhanh2_Hoan_Thanh" := "AI_PLC2_State" = 40;
END_REGION

REGION Network 107: Bản đồ trạng thái - Bồn 3 đã xả xong
   RUNG wire#powerrail
      { S7_Templates := "SrcType := Int" } EQ_Contact(in1 := "AI_PLC2_State", in2 := 15)
      { S7_Templates := "SrcType := Real" } LE_Contact(in1 := "AI_LT3213_Bon3_Eff", in2 := 0.5)
      Coil( "AI_PLC2_Xa_Bon3_Xong" )
   END_RUNG
   // the same network as SCL:
   "AI_PLC2_Xa_Bon3_Xong" := ("AI_PLC2_State" = 15) AND ("AI_LT3213_Bon3_Eff" <= 0.5);
END_REGION

REGION Network 108: Bản đồ trạng thái - Bồn 4 đã xả xong
   RUNG wire#powerrail
      { S7_Templates := "SrcType := Int" } EQ_Contact(in1 := "AI_PLC2_State", in2 := 40)
      { S7_Templates := "SrcType := Real" } LE_Contact(in1 := "AI_LT3218_Bon4_Eff", in2 := 0.5)
      Coil( "AI_PLC2_Xa_Bon4_Xong" )
   END_RUNG
   // the same network as SCL:
   "AI_PLC2_Xa_Bon4_Xong" := ("AI_PLC2_State" = 40) AND ("AI_LT3218_Bon4_Eff" <= 0.5);
END_REGION

REGION Network 109: Chuyển về Idle - Reset Auto Enable PLC2 khi xả xong
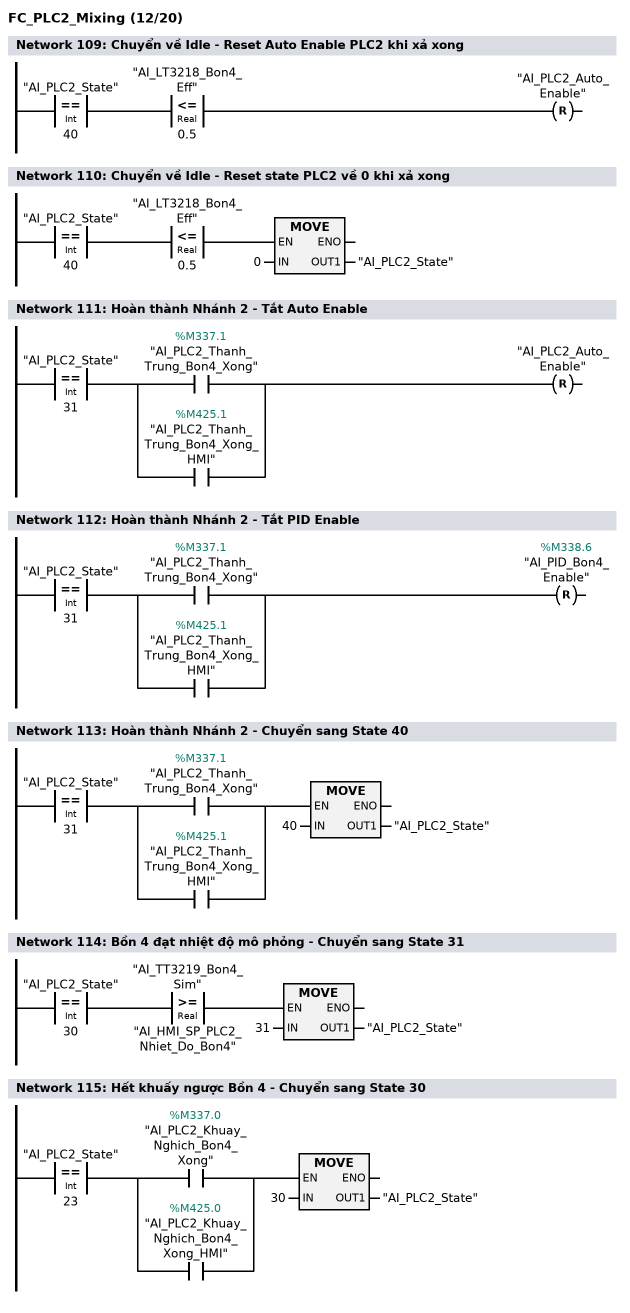
   RUNG wire#powerrail
      { S7_Templates := "SrcType := Int" } EQ_Contact(in1 := "AI_PLC2_State", in2 := 40)
      { S7_Templates := "SrcType := Real" } LE_Contact(in1 := "AI_LT3218_Bon4_Eff", in2 := 0.5)
      R_Coil( "AI_PLC2_Auto_Enable" )
   END_RUNG
   // the same network as SCL:
   IF ("AI_PLC2_State" = 40) AND ("AI_LT3218_Bon4_Eff" <= 0.5) THEN "AI_PLC2_Auto_Enable" := FALSE; END_IF;
END_REGION

REGION Network 110: Chuyển về Idle - Reset state PLC2 về 0 khi xả xong
   RUNG wire#powerrail
      { S7_Templates := "SrcType := Int" } EQ_Contact(in1 := "AI_PLC2_State", in2 := 40)
      { S7_Templates := "SrcType := Real" } LE_Contact(in1 := "AI_LT3218_Bon4_Eff", in2 := 0.5)
      { S7_GenerateENO := "TRUE" } Move(in := 0, out1 => "AI_PLC2_State")
   END_RUNG
   // the same network as SCL:
   IF ("AI_PLC2_State" = 40) AND ("AI_LT3218_Bon4_Eff" <= 0.5) THEN "AI_PLC2_State" := 0; END_IF;
END_REGION

REGION Network 111: Hoàn thành Nhánh 2 - Tắt Auto Enable
   RUNG wire#powerrail
      { S7_Templates := "SrcType := Int" } EQ_Contact(in1 := "AI_PLC2_State", in2 := 31)
      wire#w1
      Contact( "AI_PLC2_Thanh_Trung_Bon4_Xong" )
      wire#w2
      R_Coil( "AI_PLC2_Auto_Enable" )
   END_RUNG
   RUNG wire#w1
      Contact( "AI_PLC2_Thanh_Trung_Bon4_Xong_HMI" )
   END_RUNG wire#w2
   // the same network as SCL:
   IF ("AI_PLC2_State" = 31) AND ("AI_PLC2_Thanh_Trung_Bon4_Xong" OR "AI_PLC2_Thanh_Trung_Bon4_Xong_HMI") THEN
       "AI_PLC2_Auto_Enable" := FALSE;
   END_IF;
END_REGION

REGION Network 112: Hoàn thành Nhánh 2 - Tắt PID Enable
   RUNG wire#powerrail
      { S7_Templates := "SrcType := Int" } EQ_Contact(in1 := "AI_PLC2_State", in2 := 31)
      wire#w1
      Contact( "AI_PLC2_Thanh_Trung_Bon4_Xong" )
      wire#w2
      R_Coil( "AI_PID_Bon4_Enable" )
   END_RUNG
   RUNG wire#w1
      Contact( "AI_PLC2_Thanh_Trung_Bon4_Xong_HMI" )
   END_RUNG wire#w2
   // the same network as SCL:
   IF ("AI_PLC2_State" = 31) AND ("AI_PLC2_Thanh_Trung_Bon4_Xong" OR "AI_PLC2_Thanh_Trung_Bon4_Xong_HMI") THEN
       "AI_PID_Bon4_Enable" := FALSE;
   END_IF;
END_REGION

REGION Network 113: Hoàn thành Nhánh 2 - Chuyển sang State 40
   RUNG wire#powerrail
      { S7_Templates := "SrcType := Int" } EQ_Contact(in1 := "AI_PLC2_State", in2 := 31)
      wire#w1
      Contact( "AI_PLC2_Thanh_Trung_Bon4_Xong" )
      wire#w2
      { S7_GenerateENO := "TRUE" } Move(in := 40, out1 => "AI_PLC2_State")
   END_RUNG
   RUNG wire#w1
      Contact( "AI_PLC2_Thanh_Trung_Bon4_Xong_HMI" )
   END_RUNG wire#w2
   // the same network as SCL:
   IF ("AI_PLC2_State" = 31) AND ("AI_PLC2_Thanh_Trung_Bon4_Xong" OR "AI_PLC2_Thanh_Trung_Bon4_Xong_HMI") THEN
       "AI_PLC2_State" := 40;
   END_IF;
END_REGION

REGION Network 114: Bồn 4 đạt nhiệt độ mô phỏng - Chuyển sang State 31
   RUNG wire#powerrail
      { S7_Templates := "SrcType := Int" } EQ_Contact(in1 := "AI_PLC2_State", in2 := 30)
      { S7_Templates := "SrcType := Real" } GE_Contact(in1 := "AI_TT3219_Bon4_Sim", in2 := "AI_HMI_SP_PLC2_Nhiet_Do_Bon4")
      { S7_GenerateENO := "TRUE" } Move(in := 31, out1 => "AI_PLC2_State")
   END_RUNG
   // the same network as SCL:
   IF ("AI_PLC2_State" = 30) AND ("AI_TT3219_Bon4_Sim" >= "AI_HMI_SP_PLC2_Nhiet_Do_Bon4") THEN
       "AI_PLC2_State" := 31;
   END_IF;
END_REGION

REGION Network 115: Hết khuấy ngược Bồn 4 - Chuyển sang State 30
   RUNG wire#powerrail
      { S7_Templates := "SrcType := Int" } EQ_Contact(in1 := "AI_PLC2_State", in2 := 23)
      wire#w1
      Contact( "AI_PLC2_Khuay_Nghich_Bon4_Xong" )
      wire#w2
      { S7_GenerateENO := "TRUE" } Move(in := 30, out1 => "AI_PLC2_State")
   END_RUNG
   RUNG wire#w1
      Contact( "AI_PLC2_Khuay_Nghich_Bon4_Xong_HMI" )
   END_RUNG wire#w2
   // the same network as SCL:
   IF ("AI_PLC2_State" = 23) AND ("AI_PLC2_Khuay_Nghich_Bon4_Xong" OR "AI_PLC2_Khuay_Nghich_Bon4_Xong_HMI") THEN
       "AI_PLC2_State" := 30;
   END_IF;
END_REGION

REGION Network 116: Hết khuấy thuận Bồn 4 - Chuyển sang State 23
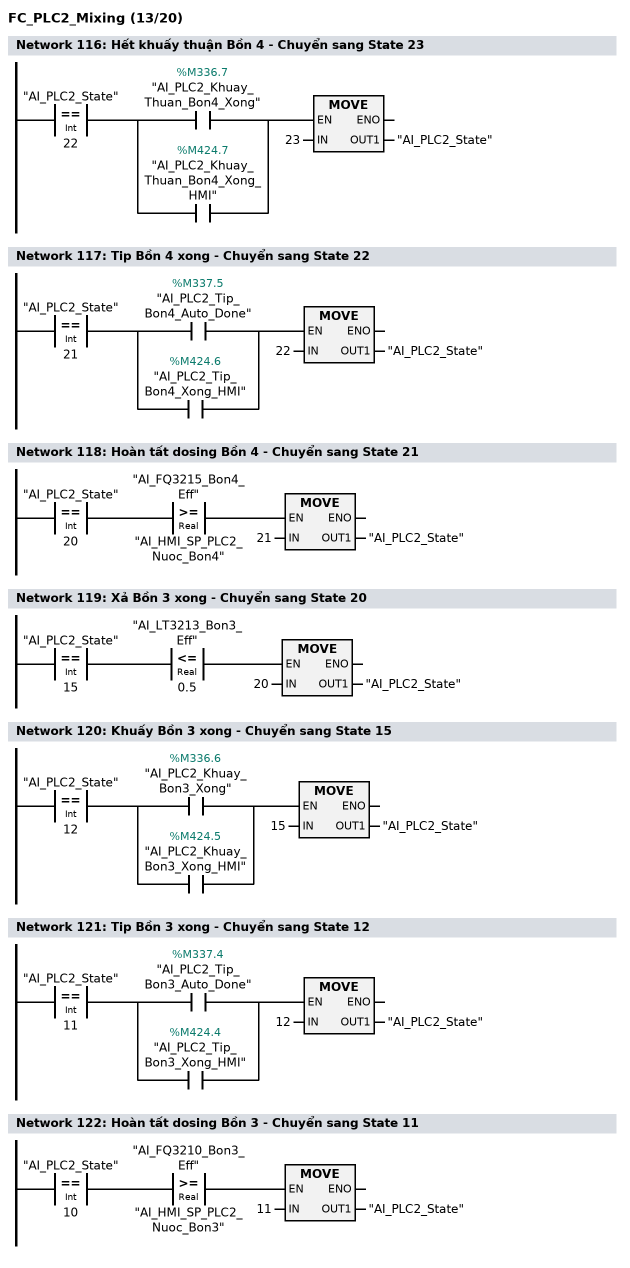
   RUNG wire#powerrail
      { S7_Templates := "SrcType := Int" } EQ_Contact(in1 := "AI_PLC2_State", in2 := 22)
      wire#w1
      Contact( "AI_PLC2_Khuay_Thuan_Bon4_Xong" )
      wire#w2
      { S7_GenerateENO := "TRUE" } Move(in := 23, out1 => "AI_PLC2_State")
   END_RUNG
   RUNG wire#w1
      Contact( "AI_PLC2_Khuay_Thuan_Bon4_Xong_HMI" )
   END_RUNG wire#w2
   // the same network as SCL:
   IF ("AI_PLC2_State" = 22) AND ("AI_PLC2_Khuay_Thuan_Bon4_Xong" OR "AI_PLC2_Khuay_Thuan_Bon4_Xong_HMI") THEN
       "AI_PLC2_State" := 23;
   END_IF;
END_REGION

REGION Network 117: Tip Bồn 4 xong - Chuyển sang State 22
   RUNG wire#powerrail
      { S7_Templates := "SrcType := Int" } EQ_Contact(in1 := "AI_PLC2_State", in2 := 21)
      wire#w1
      Contact( "AI_PLC2_Tip_Bon4_Auto_Done" )
      wire#w2
      { S7_GenerateENO := "TRUE" } Move(in := 22, out1 => "AI_PLC2_State")
   END_RUNG
   RUNG wire#w1
      Contact( "AI_PLC2_Tip_Bon4_Xong_HMI" )
   END_RUNG wire#w2
   // the same network as SCL:
   IF ("AI_PLC2_State" = 21) AND ("AI_PLC2_Tip_Bon4_Auto_Done" OR "AI_PLC2_Tip_Bon4_Xong_HMI") THEN
       "AI_PLC2_State" := 22;
   END_IF;
END_REGION

REGION Network 118: Hoàn tất dosing Bồn 4 - Chuyển sang State 21
   RUNG wire#powerrail
      { S7_Templates := "SrcType := Int" } EQ_Contact(in1 := "AI_PLC2_State", in2 := 20)
      { S7_Templates := "SrcType := Real" } GE_Contact(in1 := "AI_FQ3215_Bon4_Eff", in2 := "AI_HMI_SP_PLC2_Nuoc_Bon4")
      { S7_GenerateENO := "TRUE" } Move(in := 21, out1 => "AI_PLC2_State")
   END_RUNG
   // the same network as SCL:
   IF ("AI_PLC2_State" = 20) AND ("AI_FQ3215_Bon4_Eff" >= "AI_HMI_SP_PLC2_Nuoc_Bon4") THEN
       "AI_PLC2_State" := 21;
   END_IF;
END_REGION

REGION Network 119: Xả Bồn 3 xong - Chuyển sang State 20
   RUNG wire#powerrail
      { S7_Templates := "SrcType := Int" } EQ_Contact(in1 := "AI_PLC2_State", in2 := 15)
      { S7_Templates := "SrcType := Real" } LE_Contact(in1 := "AI_LT3213_Bon3_Eff", in2 := 0.5)
      { S7_GenerateENO := "TRUE" } Move(in := 20, out1 => "AI_PLC2_State")
   END_RUNG
   // the same network as SCL:
   IF ("AI_PLC2_State" = 15) AND ("AI_LT3213_Bon3_Eff" <= 0.5) THEN "AI_PLC2_State" := 20; END_IF;
END_REGION

REGION Network 120: Khuấy Bồn 3 xong - Chuyển sang State 15
   RUNG wire#powerrail
      { S7_Templates := "SrcType := Int" } EQ_Contact(in1 := "AI_PLC2_State", in2 := 12)
      wire#w1
      Contact( "AI_PLC2_Khuay_Bon3_Xong" )
      wire#w2
      { S7_GenerateENO := "TRUE" } Move(in := 15, out1 => "AI_PLC2_State")
   END_RUNG
   RUNG wire#w1
      Contact( "AI_PLC2_Khuay_Bon3_Xong_HMI" )
   END_RUNG wire#w2
   // the same network as SCL:
   IF ("AI_PLC2_State" = 12) AND ("AI_PLC2_Khuay_Bon3_Xong" OR "AI_PLC2_Khuay_Bon3_Xong_HMI") THEN
       "AI_PLC2_State" := 15;
   END_IF;
END_REGION

REGION Network 121: Tip Bồn 3 xong - Chuyển sang State 12
   RUNG wire#powerrail
      { S7_Templates := "SrcType := Int" } EQ_Contact(in1 := "AI_PLC2_State", in2 := 11)
      wire#w1
      Contact( "AI_PLC2_Tip_Bon3_Auto_Done" )
      wire#w2
      { S7_GenerateENO := "TRUE" } Move(in := 12, out1 => "AI_PLC2_State")
   END_RUNG
   RUNG wire#w1
      Contact( "AI_PLC2_Tip_Bon3_Xong_HMI" )
   END_RUNG wire#w2
   // the same network as SCL:
   IF ("AI_PLC2_State" = 11) AND ("AI_PLC2_Tip_Bon3_Auto_Done" OR "AI_PLC2_Tip_Bon3_Xong_HMI") THEN
       "AI_PLC2_State" := 12;
   END_IF;
END_REGION

REGION Network 122: Hoàn tất dosing Bồn 3 - Chuyển sang State 11
   RUNG wire#powerrail
      { S7_Templates := "SrcType := Int" } EQ_Contact(in1 := "AI_PLC2_State", in2 := 10)
      { S7_Templates := "SrcType := Real" } GE_Contact(in1 := "AI_FQ3210_Bon3_Eff", in2 := "AI_HMI_SP_PLC2_Nuoc_Bon3")
      { S7_GenerateENO := "TRUE" } Move(in := 11, out1 => "AI_PLC2_State")
   END_RUNG
   // the same network as SCL:
   IF ("AI_PLC2_State" = 10) AND ("AI_FQ3210_Bon3_Eff" >= "AI_HMI_SP_PLC2_Nuoc_Bon3") THEN
       "AI_PLC2_State" := 11;
   END_IF;
END_REGION

REGION Network 123: Timer đếm thời gian Tip Bồn 3
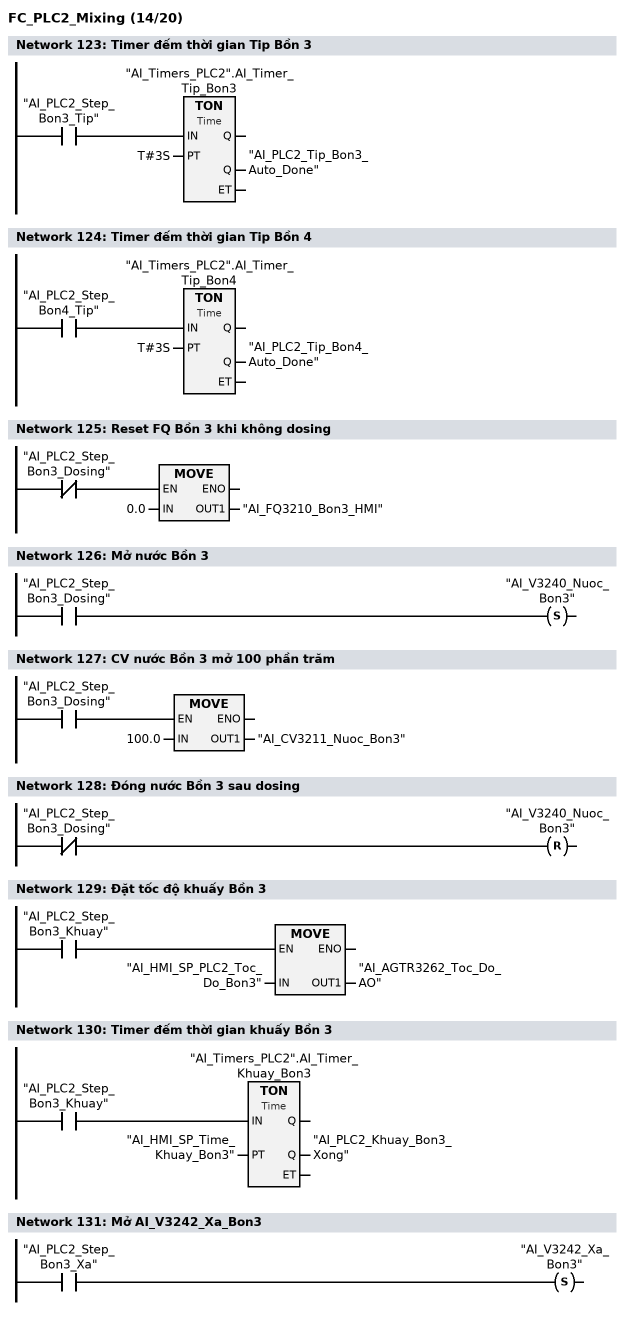
   RUNG wire#powerrail
      Contact( "AI_PLC2_Step_Bon3_Tip" )
      { S7_Templates := "time_type := Time" } "AI_Timers_PLC2".AI_Timer_Tip_Bon3.TON(pt := T#3S, q => "AI_PLC2_Tip_Bon3_Auto_Done", et =>)
   END_RUNG
   // the same network as SCL:
   "AI_Timers_PLC2".AI_Timer_Tip_Bon3.TON(IN := "AI_PLC2_Step_Bon3_Tip",
                           PT := T#3S,
                           Q => "AI_PLC2_Tip_Bon3_Auto_Done");
END_REGION

REGION Network 124: Timer đếm thời gian Tip Bồn 4
   RUNG wire#powerrail
      Contact( "AI_PLC2_Step_Bon4_Tip" )
      { S7_Templates := "time_type := Time" } "AI_Timers_PLC2".AI_Timer_Tip_Bon4.TON(pt := T#3S, q => "AI_PLC2_Tip_Bon4_Auto_Done", et =>)
   END_RUNG
   // the same network as SCL:
   "AI_Timers_PLC2".AI_Timer_Tip_Bon4.TON(IN := "AI_PLC2_Step_Bon4_Tip",
                           PT := T#3S,
                           Q => "AI_PLC2_Tip_Bon4_Auto_Done");
END_REGION

REGION Network 125: Reset FQ Bồn 3 khi không dosing
   RUNG wire#powerrail
      I_Contact( "AI_PLC2_Step_Bon3_Dosing" )
      { S7_GenerateENO := "TRUE" } Move(in := 0.0, out1 => "AI_FQ3210_Bon3_HMI")
   END_RUNG
   // the same network as SCL:
   IF NOT "AI_PLC2_Step_Bon3_Dosing" THEN "AI_FQ3210_Bon3_HMI" := 0.0; END_IF;
END_REGION

REGION Network 126: Mở nước Bồn 3
   RUNG wire#powerrail
      Contact( "AI_PLC2_Step_Bon3_Dosing" )
      S_Coil( "AI_V3240_Nuoc_Bon3" )
   END_RUNG
   // the same network as SCL:
   IF "AI_PLC2_Step_Bon3_Dosing" THEN "AI_V3240_Nuoc_Bon3" := TRUE; END_IF;
END_REGION

REGION Network 127: CV nước Bồn 3 mở 100 phần trăm
   RUNG wire#powerrail
      Contact( "AI_PLC2_Step_Bon3_Dosing" )
      { S7_GenerateENO := "TRUE" } Move(in := 100.0, out1 => "AI_CV3211_Nuoc_Bon3")
   END_RUNG
   // the same network as SCL:
   IF "AI_PLC2_Step_Bon3_Dosing" THEN "AI_CV3211_Nuoc_Bon3" := 100.0; END_IF;
END_REGION

REGION Network 128: Đóng nước Bồn 3 sau dosing
   RUNG wire#powerrail
      I_Contact( "AI_PLC2_Step_Bon3_Dosing" )
      R_Coil( "AI_V3240_Nuoc_Bon3" )
   END_RUNG
   // the same network as SCL:
   IF NOT "AI_PLC2_Step_Bon3_Dosing" THEN "AI_V3240_Nuoc_Bon3" := FALSE; END_IF;
END_REGION

REGION Network 129: Đặt tốc độ khuấy Bồn 3
   RUNG wire#powerrail
      Contact( "AI_PLC2_Step_Bon3_Khuay" )
      { S7_GenerateENO := "TRUE" } Move(in := "AI_HMI_SP_PLC2_Toc_Do_Bon3", out1 => "AI_AGTR3262_Toc_Do_AO")
   END_RUNG
   // the same network as SCL:
   IF "AI_PLC2_Step_Bon3_Khuay" THEN "AI_AGTR3262_Toc_Do_AO" := "AI_HMI_SP_PLC2_Toc_Do_Bon3"; END_IF;
END_REGION

REGION Network 130: Timer đếm thời gian khuấy Bồn 3
   RUNG wire#powerrail
      Contact( "AI_PLC2_Step_Bon3_Khuay" )
      { S7_Templates := "time_type := Time" } "AI_Timers_PLC2".AI_Timer_Khuay_Bon3.TON(pt := "AI_HMI_SP_Time_Khuay_Bon3", q => "AI_PLC2_Khuay_Bon3_Xong", et =>)
   END_RUNG
   // the same network as SCL:
   "AI_Timers_PLC2".AI_Timer_Khuay_Bon3.TON(IN := "AI_PLC2_Step_Bon3_Khuay",
                           PT := "AI_HMI_SP_Time_Khuay_Bon3",
                           Q => "AI_PLC2_Khuay_Bon3_Xong");
END_REGION

REGION Network 131: Mở AI_V3242_Xa_Bon3
   RUNG wire#powerrail
      Contact( "AI_PLC2_Step_Bon3_Xa" )
      S_Coil( "AI_V3242_Xa_Bon3" )
   END_RUNG
   // the same network as SCL:
   IF "AI_PLC2_Step_Bon3_Xa" THEN "AI_V3242_Xa_Bon3" := TRUE; END_IF;
END_REGION

REGION Network 132: Mở AI_V3243_Xa_Bon3
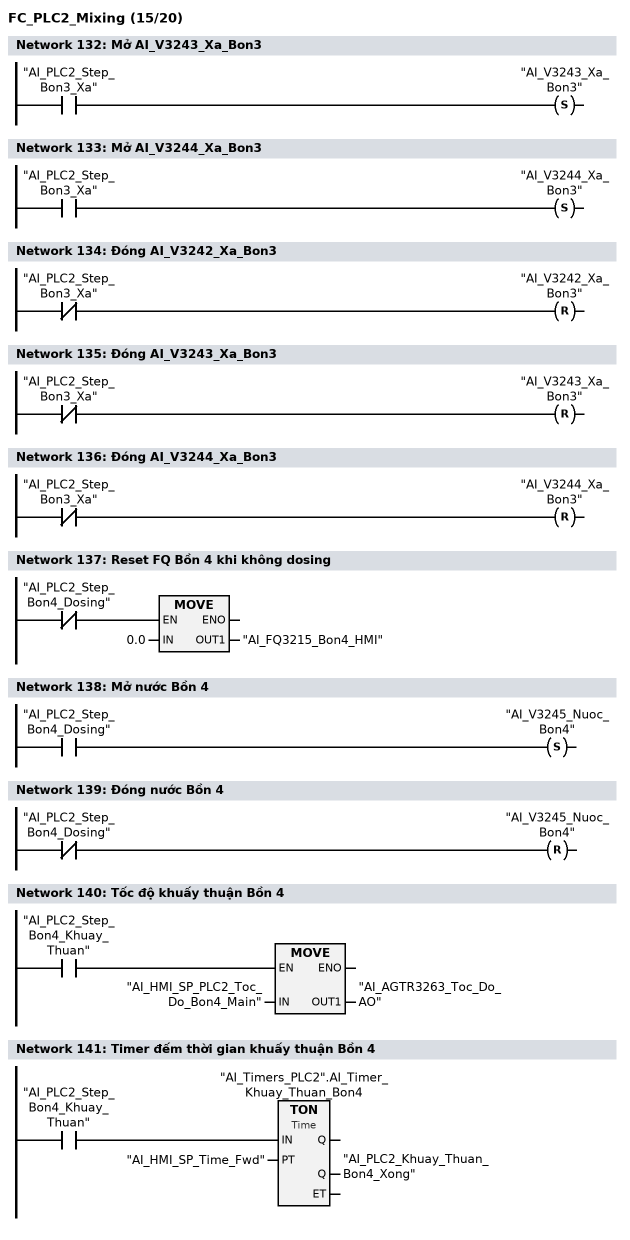
   RUNG wire#powerrail
      Contact( "AI_PLC2_Step_Bon3_Xa" )
      S_Coil( "AI_V3243_Xa_Bon3" )
   END_RUNG
   // the same network as SCL:
   IF "AI_PLC2_Step_Bon3_Xa" THEN "AI_V3243_Xa_Bon3" := TRUE; END_IF;
END_REGION

REGION Network 133: Mở AI_V3244_Xa_Bon3
   RUNG wire#powerrail
      Contact( "AI_PLC2_Step_Bon3_Xa" )
      S_Coil( "AI_V3244_Xa_Bon3" )
   END_RUNG
   // the same network as SCL:
   IF "AI_PLC2_Step_Bon3_Xa" THEN "AI_V3244_Xa_Bon3" := TRUE; END_IF;
END_REGION

REGION Network 134: Đóng AI_V3242_Xa_Bon3
   RUNG wire#powerrail
      I_Contact( "AI_PLC2_Step_Bon3_Xa" )
      R_Coil( "AI_V3242_Xa_Bon3" )
   END_RUNG
   // the same network as SCL:
   IF NOT "AI_PLC2_Step_Bon3_Xa" THEN "AI_V3242_Xa_Bon3" := FALSE; END_IF;
END_REGION

REGION Network 135: Đóng AI_V3243_Xa_Bon3
   RUNG wire#powerrail
      I_Contact( "AI_PLC2_Step_Bon3_Xa" )
      R_Coil( "AI_V3243_Xa_Bon3" )
   END_RUNG
   // the same network as SCL:
   IF NOT "AI_PLC2_Step_Bon3_Xa" THEN "AI_V3243_Xa_Bon3" := FALSE; END_IF;
END_REGION

REGION Network 136: Đóng AI_V3244_Xa_Bon3
   RUNG wire#powerrail
      I_Contact( "AI_PLC2_Step_Bon3_Xa" )
      R_Coil( "AI_V3244_Xa_Bon3" )
   END_RUNG
   // the same network as SCL:
   IF NOT "AI_PLC2_Step_Bon3_Xa" THEN "AI_V3244_Xa_Bon3" := FALSE; END_IF;
END_REGION

REGION Network 137: Reset FQ Bồn 4 khi không dosing
   RUNG wire#powerrail
      I_Contact( "AI_PLC2_Step_Bon4_Dosing" )
      { S7_GenerateENO := "TRUE" } Move(in := 0.0, out1 => "AI_FQ3215_Bon4_HMI")
   END_RUNG
   // the same network as SCL:
   IF NOT "AI_PLC2_Step_Bon4_Dosing" THEN "AI_FQ3215_Bon4_HMI" := 0.0; END_IF;
END_REGION

REGION Network 138: Mở nước Bồn 4
   RUNG wire#powerrail
      Contact( "AI_PLC2_Step_Bon4_Dosing" )
      S_Coil( "AI_V3245_Nuoc_Bon4" )
   END_RUNG
   // the same network as SCL:
   IF "AI_PLC2_Step_Bon4_Dosing" THEN "AI_V3245_Nuoc_Bon4" := TRUE; END_IF;
END_REGION

REGION Network 139: Đóng nước Bồn 4
   RUNG wire#powerrail
      I_Contact( "AI_PLC2_Step_Bon4_Dosing" )
      R_Coil( "AI_V3245_Nuoc_Bon4" )
   END_RUNG
   // the same network as SCL:
   IF NOT "AI_PLC2_Step_Bon4_Dosing" THEN "AI_V3245_Nuoc_Bon4" := FALSE; END_IF;
END_REGION

REGION Network 140: Tốc độ khuấy thuận Bồn 4
   RUNG wire#powerrail
      Contact( "AI_PLC2_Step_Bon4_Khuay_Thuan" )
      { S7_GenerateENO := "TRUE" } Move(in := "AI_HMI_SP_PLC2_Toc_Do_Bon4_Main", out1 => "AI_AGTR3263_Toc_Do_AO")
   END_RUNG
   // the same network as SCL:
   IF "AI_PLC2_Step_Bon4_Khuay_Thuan" THEN
       "AI_AGTR3263_Toc_Do_AO" := "AI_HMI_SP_PLC2_Toc_Do_Bon4_Main";
   END_IF;
END_REGION

REGION Network 141: Timer đếm thời gian khuấy thuận Bồn 4
   RUNG wire#powerrail
      Contact( "AI_PLC2_Step_Bon4_Khuay_Thuan" )
      { S7_Templates := "time_type := Time" } "AI_Timers_PLC2".AI_Timer_Khuay_Thuan_Bon4.TON(pt := "AI_HMI_SP_Time_Fwd", q => "AI_PLC2_Khuay_Thuan_Bon4_Xong", et =>)
   END_RUNG
   // the same network as SCL:
   "AI_Timers_PLC2".AI_Timer_Khuay_Thuan_Bon4.TON(IN := "AI_PLC2_Step_Bon4_Khuay_Thuan",
                           PT := "AI_HMI_SP_Time_Fwd",
                           Q => "AI_PLC2_Khuay_Thuan_Bon4_Xong");
END_REGION

REGION Network 142: Timer đếm thời gian khuấy ngược Bồn 4
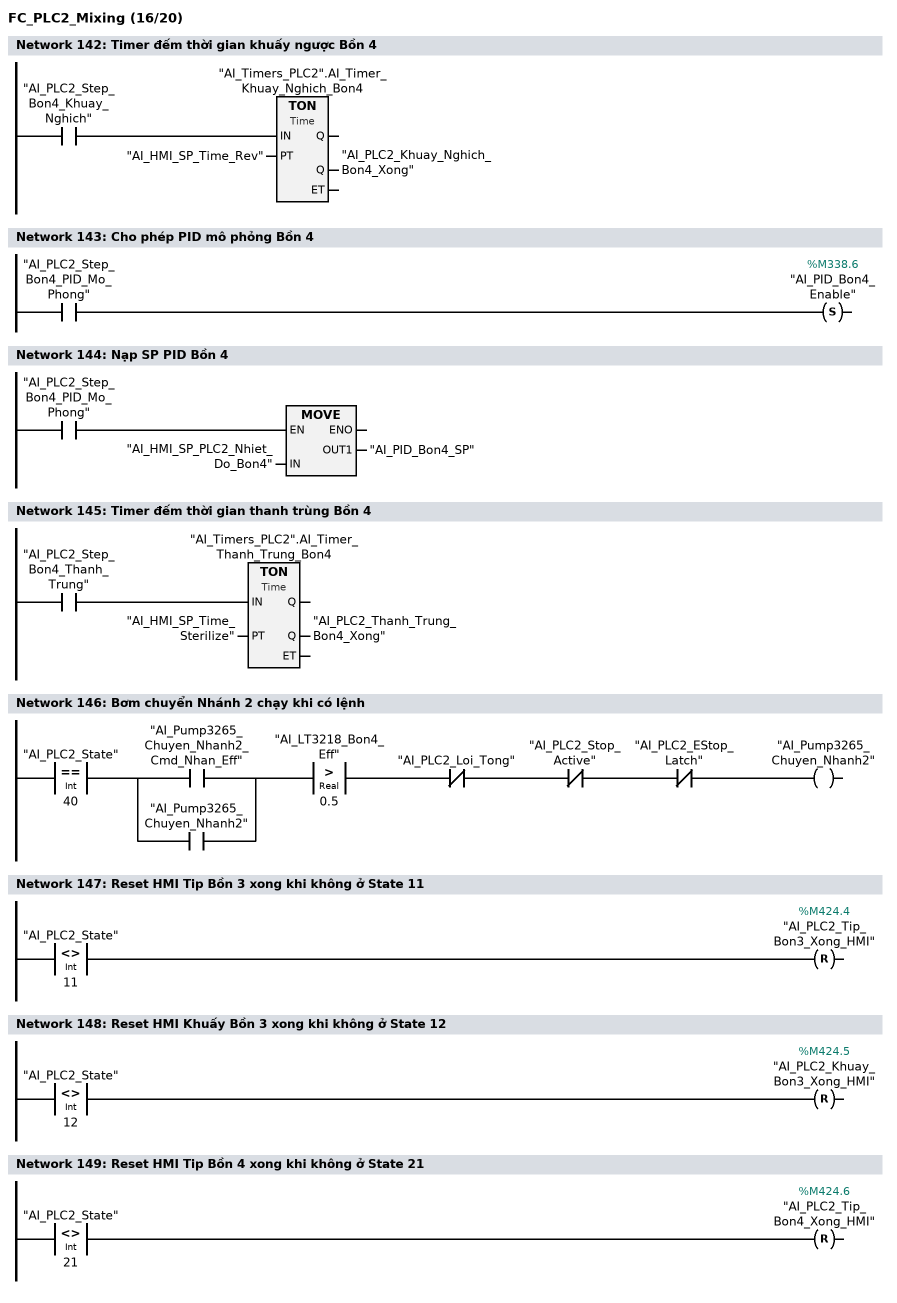
   RUNG wire#powerrail
      Contact( "AI_PLC2_Step_Bon4_Khuay_Nghich" )
      { S7_Templates := "time_type := Time" } "AI_Timers_PLC2".AI_Timer_Khuay_Nghich_Bon4.TON(pt := "AI_HMI_SP_Time_Rev", q => "AI_PLC2_Khuay_Nghich_Bon4_Xong", et =>)
   END_RUNG
   // the same network as SCL:
   "AI_Timers_PLC2".AI_Timer_Khuay_Nghich_Bon4.TON(IN := "AI_PLC2_Step_Bon4_Khuay_Nghich",
                           PT := "AI_HMI_SP_Time_Rev",
                           Q => "AI_PLC2_Khuay_Nghich_Bon4_Xong");
END_REGION

REGION Network 143: Cho phép PID mô phỏng Bồn 4
   RUNG wire#powerrail
      Contact( "AI_PLC2_Step_Bon4_PID_Mo_Phong" )
      S_Coil( "AI_PID_Bon4_Enable" )
   END_RUNG
   // the same network as SCL:
   IF "AI_PLC2_Step_Bon4_PID_Mo_Phong" THEN "AI_PID_Bon4_Enable" := TRUE; END_IF;
END_REGION

REGION Network 144: Nạp SP PID Bồn 4
   RUNG wire#powerrail
      Contact( "AI_PLC2_Step_Bon4_PID_Mo_Phong" )
      { S7_GenerateENO := "TRUE" } Move(in := "AI_HMI_SP_PLC2_Nhiet_Do_Bon4", out1 => "AI_PID_Bon4_SP")
   END_RUNG
   // the same network as SCL:
   IF "AI_PLC2_Step_Bon4_PID_Mo_Phong" THEN "AI_PID_Bon4_SP" := "AI_HMI_SP_PLC2_Nhiet_Do_Bon4"; END_IF;
END_REGION

REGION Network 145: Timer đếm thời gian thanh trùng Bồn 4
   RUNG wire#powerrail
      Contact( "AI_PLC2_Step_Bon4_Thanh_Trung" )
      { S7_Templates := "time_type := Time" } "AI_Timers_PLC2".AI_Timer_Thanh_Trung_Bon4.TON(pt := "AI_HMI_SP_Time_Sterilize", q => "AI_PLC2_Thanh_Trung_Bon4_Xong", et =>)
   END_RUNG
   // the same network as SCL:
   "AI_Timers_PLC2".AI_Timer_Thanh_Trung_Bon4.TON(IN := "AI_PLC2_Step_Bon4_Thanh_Trung",
                           PT := "AI_HMI_SP_Time_Sterilize",
                           Q => "AI_PLC2_Thanh_Trung_Bon4_Xong");
END_REGION

REGION Network 146: Bơm chuyển Nhánh 2 chạy khi có lệnh
   RUNG wire#powerrail
      { S7_Templates := "SrcType := Int" } EQ_Contact(in1 := "AI_PLC2_State", in2 := 40)
      wire#w1
      Contact( "AI_Pump3265_Chuyen_Nhanh2_Cmd_Nhan_Eff" )
      wire#w2
      { S7_Templates := "SrcType := Real" } GT_Contact(in1 := "AI_LT3218_Bon4_Eff", in2 := 0.5)
      I_Contact( "AI_PLC2_Loi_Tong" )
      I_Contact( "AI_PLC2_Stop_Active" )
      I_Contact( "AI_PLC2_EStop_Latch" )
      Coil( "AI_Pump3265_Chuyen_Nhanh2" )
   END_RUNG
   RUNG wire#w1
      Contact( "AI_Pump3265_Chuyen_Nhanh2" )
   END_RUNG wire#w2
   // the same network as SCL:
   "AI_Pump3265_Chuyen_Nhanh2" := ("AI_PLC2_State" = 40) AND ("AI_Pump3265_Chuyen_Nhanh2_Cmd_Nhan_Eff" OR "AI_Pump3265_Chuyen_Nhanh2") AND ("AI_LT3218_Bon4_Eff" > 0.5) AND NOT "AI_PLC2_Loi_Tong" AND NOT "AI_PLC2_Stop_Active" AND NOT "AI_PLC2_EStop_Latch";
END_REGION

REGION Network 147: Reset HMI Tip Bồn 3 xong khi không ở State 11
   RUNG wire#powerrail
      { S7_Templates := "SrcType := Int" } NE_Contact(in1 := "AI_PLC2_State", in2 := 11)
      R_Coil( "AI_PLC2_Tip_Bon3_Xong_HMI" )
   END_RUNG
   // the same network as SCL:
   IF "AI_PLC2_State" <> 11 THEN "AI_PLC2_Tip_Bon3_Xong_HMI" := FALSE; END_IF;
END_REGION

REGION Network 148: Reset HMI Khuấy Bồn 3 xong khi không ở State 12
   RUNG wire#powerrail
      { S7_Templates := "SrcType := Int" } NE_Contact(in1 := "AI_PLC2_State", in2 := 12)
      R_Coil( "AI_PLC2_Khuay_Bon3_Xong_HMI" )
   END_RUNG
   // the same network as SCL:
   IF "AI_PLC2_State" <> 12 THEN "AI_PLC2_Khuay_Bon3_Xong_HMI" := FALSE; END_IF;
END_REGION

REGION Network 149: Reset HMI Tip Bồn 4 xong khi không ở State 21
   RUNG wire#powerrail
      { S7_Templates := "SrcType := Int" } NE_Contact(in1 := "AI_PLC2_State", in2 := 21)
      R_Coil( "AI_PLC2_Tip_Bon4_Xong_HMI" )
   END_RUNG
   // the same network as SCL:
   IF "AI_PLC2_State" <> 21 THEN "AI_PLC2_Tip_Bon4_Xong_HMI" := FALSE; END_IF;
END_REGION

REGION Network 150: Reset HMI Khuấy thuận Bồn 4 xong khi không ở State 22
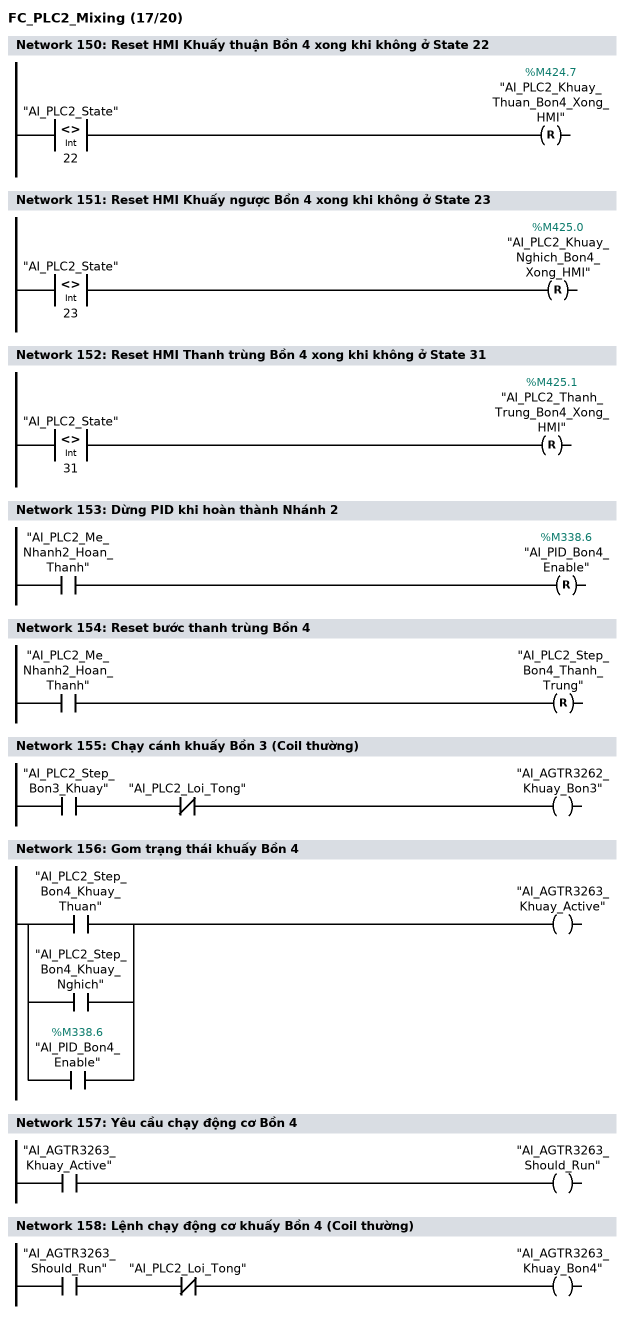
   RUNG wire#powerrail
      { S7_Templates := "SrcType := Int" } NE_Contact(in1 := "AI_PLC2_State", in2 := 22)
      R_Coil( "AI_PLC2_Khuay_Thuan_Bon4_Xong_HMI" )
   END_RUNG
   // the same network as SCL:
   IF "AI_PLC2_State" <> 22 THEN "AI_PLC2_Khuay_Thuan_Bon4_Xong_HMI" := FALSE; END_IF;
END_REGION

REGION Network 151: Reset HMI Khuấy ngược Bồn 4 xong khi không ở State 23
   RUNG wire#powerrail
      { S7_Templates := "SrcType := Int" } NE_Contact(in1 := "AI_PLC2_State", in2 := 23)
      R_Coil( "AI_PLC2_Khuay_Nghich_Bon4_Xong_HMI" )
   END_RUNG
   // the same network as SCL:
   IF "AI_PLC2_State" <> 23 THEN "AI_PLC2_Khuay_Nghich_Bon4_Xong_HMI" := FALSE; END_IF;
END_REGION

REGION Network 152: Reset HMI Thanh trùng Bồn 4 xong khi không ở State 31
   RUNG wire#powerrail
      { S7_Templates := "SrcType := Int" } NE_Contact(in1 := "AI_PLC2_State", in2 := 31)
      R_Coil( "AI_PLC2_Thanh_Trung_Bon4_Xong_HMI" )
   END_RUNG
   // the same network as SCL:
   IF "AI_PLC2_State" <> 31 THEN "AI_PLC2_Thanh_Trung_Bon4_Xong_HMI" := FALSE; END_IF;
END_REGION

REGION Network 153: Dừng PID khi hoàn thành Nhánh 2
   RUNG wire#powerrail
      Contact( "AI_PLC2_Me_Nhanh2_Hoan_Thanh" )
      R_Coil( "AI_PID_Bon4_Enable" )
   END_RUNG
   // the same network as SCL:
   IF "AI_PLC2_Me_Nhanh2_Hoan_Thanh" THEN "AI_PID_Bon4_Enable" := FALSE; END_IF;
END_REGION

REGION Network 154: Reset bước thanh trùng Bồn 4
   RUNG wire#powerrail
      Contact( "AI_PLC2_Me_Nhanh2_Hoan_Thanh" )
      R_Coil( "AI_PLC2_Step_Bon4_Thanh_Trung" )
   END_RUNG
   // the same network as SCL:
   IF "AI_PLC2_Me_Nhanh2_Hoan_Thanh" THEN "AI_PLC2_Step_Bon4_Thanh_Trung" := FALSE; END_IF;
END_REGION

REGION Network 155: Chạy cánh khuấy Bồn 3 (Coil thường)
   RUNG wire#powerrail
      Contact( "AI_PLC2_Step_Bon3_Khuay" )
      I_Contact( "AI_PLC2_Loi_Tong" )
      Coil( "AI_AGTR3262_Khuay_Bon3" )
   END_RUNG
   // the same network as SCL:
   "AI_AGTR3262_Khuay_Bon3" := "AI_PLC2_Step_Bon3_Khuay" AND NOT "AI_PLC2_Loi_Tong";
END_REGION

REGION Network 156: Gom trạng thái khuấy Bồn 4
   RUNG wire#powerrail
      Contact( "AI_PLC2_Step_Bon4_Khuay_Thuan" )
      wire#w1
      Coil( "AI_AGTR3263_Khuay_Active" )
   END_RUNG
   RUNG wire#powerrail
      Contact( "AI_PLC2_Step_Bon4_Khuay_Nghich" )
   END_RUNG wire#w1
   RUNG wire#powerrail
      Contact( "AI_PID_Bon4_Enable" )
   END_RUNG wire#w1
   // the same network as SCL:
   "AI_AGTR3263_Khuay_Active" := "AI_PLC2_Step_Bon4_Khuay_Thuan" OR "AI_PLC2_Step_Bon4_Khuay_Nghich" OR "AI_PID_Bon4_Enable";
END_REGION

REGION Network 157: Yêu cầu chạy động cơ Bồn 4
   RUNG wire#powerrail
      Contact( "AI_AGTR3263_Khuay_Active" )
      Coil( "AI_AGTR3263_Should_Run" )
   END_RUNG
   // the same network as SCL:
   "AI_AGTR3263_Should_Run" := "AI_AGTR3263_Khuay_Active";
END_REGION

REGION Network 158: Lệnh chạy động cơ khuấy Bồn 4 (Coil thường)
   RUNG wire#powerrail
      Contact( "AI_AGTR3263_Should_Run" )
      I_Contact( "AI_PLC2_Loi_Tong" )
      Coil( "AI_AGTR3263_Khuay_Bon4" )
   END_RUNG
   // the same network as SCL:
   "AI_AGTR3263_Khuay_Bon4" := "AI_AGTR3263_Should_Run" AND NOT "AI_PLC2_Loi_Tong";
END_REGION

REGION Network 159: Lệnh đảo chiều động cơ khuấy Bồn 4 (Coil thường)
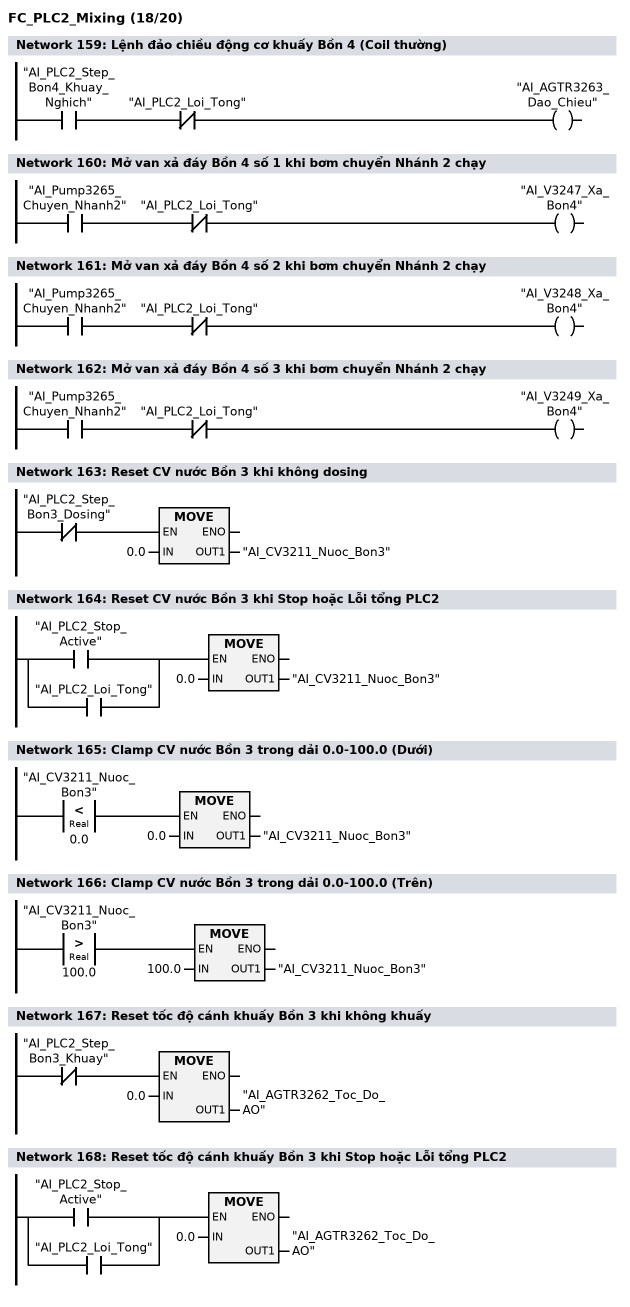
   RUNG wire#powerrail
      Contact( "AI_PLC2_Step_Bon4_Khuay_Nghich" )
      I_Contact( "AI_PLC2_Loi_Tong" )
      Coil( "AI_AGTR3263_Dao_Chieu" )
   END_RUNG
   // the same network as SCL:
   "AI_AGTR3263_Dao_Chieu" := "AI_PLC2_Step_Bon4_Khuay_Nghich" AND NOT "AI_PLC2_Loi_Tong";
END_REGION

REGION Network 160: Mở van xả đáy Bồn 4 số 1 khi bơm chuyển Nhánh 2 chạy
   RUNG wire#powerrail
      Contact( "AI_Pump3265_Chuyen_Nhanh2" )
      I_Contact( "AI_PLC2_Loi_Tong" )
      Coil( "AI_V3247_Xa_Bon4" )
   END_RUNG
   // the same network as SCL:
   "AI_V3247_Xa_Bon4" := "AI_Pump3265_Chuyen_Nhanh2" AND NOT "AI_PLC2_Loi_Tong";
END_REGION

REGION Network 161: Mở van xả đáy Bồn 4 số 2 khi bơm chuyển Nhánh 2 chạy
   RUNG wire#powerrail
      Contact( "AI_Pump3265_Chuyen_Nhanh2" )
      I_Contact( "AI_PLC2_Loi_Tong" )
      Coil( "AI_V3248_Xa_Bon4" )
   END_RUNG
   // the same network as SCL:
   "AI_V3248_Xa_Bon4" := "AI_Pump3265_Chuyen_Nhanh2" AND NOT "AI_PLC2_Loi_Tong";
END_REGION

REGION Network 162: Mở van xả đáy Bồn 4 số 3 khi bơm chuyển Nhánh 2 chạy
   RUNG wire#powerrail
      Contact( "AI_Pump3265_Chuyen_Nhanh2" )
      I_Contact( "AI_PLC2_Loi_Tong" )
      Coil( "AI_V3249_Xa_Bon4" )
   END_RUNG
   // the same network as SCL:
   "AI_V3249_Xa_Bon4" := "AI_Pump3265_Chuyen_Nhanh2" AND NOT "AI_PLC2_Loi_Tong";
END_REGION

REGION Network 163: Reset CV nước Bồn 3 khi không dosing
   RUNG wire#powerrail
      I_Contact( "AI_PLC2_Step_Bon3_Dosing" )
      { S7_GenerateENO := "TRUE" } Move(in := 0.0, out1 => "AI_CV3211_Nuoc_Bon3")
   END_RUNG
   // the same network as SCL:
   IF NOT "AI_PLC2_Step_Bon3_Dosing" THEN "AI_CV3211_Nuoc_Bon3" := 0.0; END_IF;
END_REGION

REGION Network 164: Reset CV nước Bồn 3 khi Stop hoặc Lỗi tổng PLC2
   RUNG wire#powerrail
      Contact( "AI_PLC2_Stop_Active" )
      wire#w1
      { S7_GenerateENO := "TRUE" } Move(in := 0.0, out1 => "AI_CV3211_Nuoc_Bon3")
   END_RUNG
   RUNG wire#powerrail
      Contact( "AI_PLC2_Loi_Tong" )
   END_RUNG wire#w1
   // the same network as SCL:
   IF "AI_PLC2_Stop_Active" OR "AI_PLC2_Loi_Tong" THEN "AI_CV3211_Nuoc_Bon3" := 0.0; END_IF;
END_REGION

REGION Network 165: Clamp CV nước Bồn 3 trong dải 0.0-100.0 (Dưới)
   RUNG wire#powerrail
      { S7_Templates := "SrcType := Real" } LT_Contact(in1 := "AI_CV3211_Nuoc_Bon3", in2 := 0.0)
      { S7_GenerateENO := "TRUE" } Move(in := 0.0, out1 => "AI_CV3211_Nuoc_Bon3")
   END_RUNG
   // the same network as SCL:
   IF "AI_CV3211_Nuoc_Bon3" < 0.0 THEN "AI_CV3211_Nuoc_Bon3" := 0.0; END_IF;
END_REGION

REGION Network 166: Clamp CV nước Bồn 3 trong dải 0.0-100.0 (Trên)
   RUNG wire#powerrail
      { S7_Templates := "SrcType := Real" } GT_Contact(in1 := "AI_CV3211_Nuoc_Bon3", in2 := 100.0)
      { S7_GenerateENO := "TRUE" } Move(in := 100.0, out1 => "AI_CV3211_Nuoc_Bon3")
   END_RUNG
   // the same network as SCL:
   IF "AI_CV3211_Nuoc_Bon3" > 100.0 THEN "AI_CV3211_Nuoc_Bon3" := 100.0; END_IF;
END_REGION

REGION Network 167: Reset tốc độ cánh khuấy Bồn 3 khi không khuấy
   RUNG wire#powerrail
      I_Contact( "AI_PLC2_Step_Bon3_Khuay" )
      { S7_GenerateENO := "TRUE" } Move(in := 0.0, out1 => "AI_AGTR3262_Toc_Do_AO")
   END_RUNG
   // the same network as SCL:
   IF NOT "AI_PLC2_Step_Bon3_Khuay" THEN "AI_AGTR3262_Toc_Do_AO" := 0.0; END_IF;
END_REGION

REGION Network 168: Reset tốc độ cánh khuấy Bồn 3 khi Stop hoặc Lỗi tổng PLC2
   RUNG wire#powerrail
      Contact( "AI_PLC2_Stop_Active" )
      wire#w1
      { S7_GenerateENO := "TRUE" } Move(in := 0.0, out1 => "AI_AGTR3262_Toc_Do_AO")
   END_RUNG
   RUNG wire#powerrail
      Contact( "AI_PLC2_Loi_Tong" )
   END_RUNG wire#w1
   // the same network as SCL:
   IF "AI_PLC2_Stop_Active" OR "AI_PLC2_Loi_Tong" THEN "AI_AGTR3262_Toc_Do_AO" := 0.0; END_IF;
END_REGION

REGION Network 169: Clamp tốc độ cánh khuấy Bồn 3 trong dải 0.0-100.0 (Dưới)
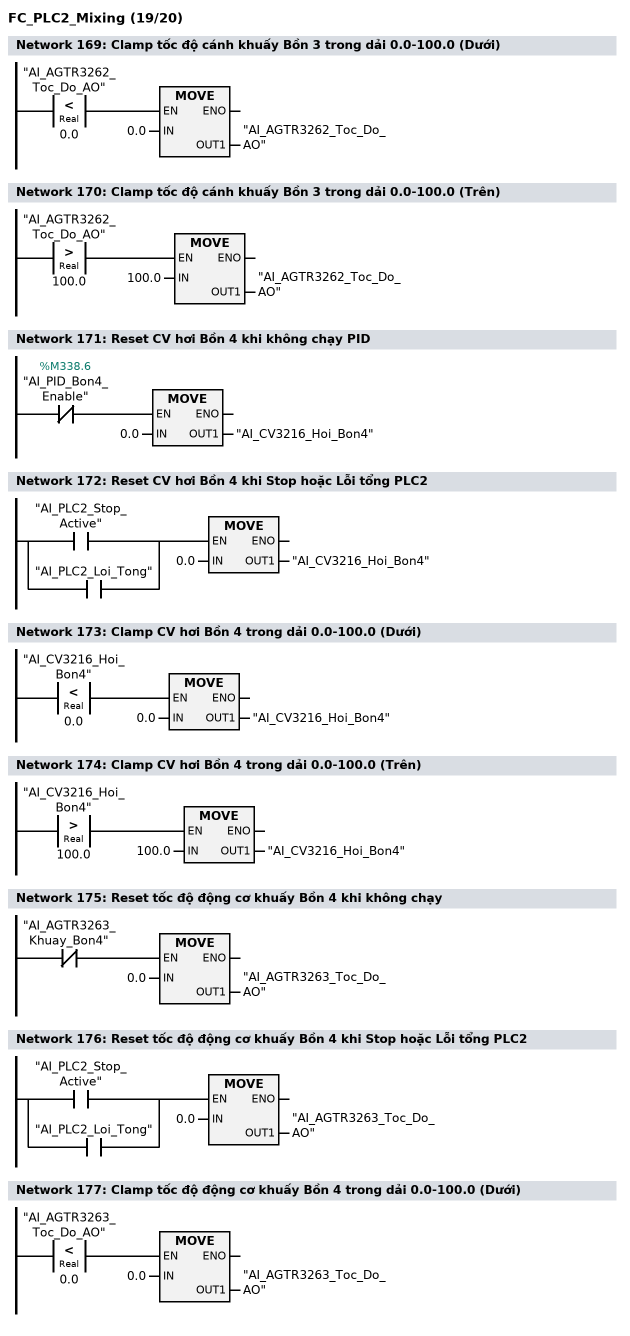
   RUNG wire#powerrail
      { S7_Templates := "SrcType := Real" } LT_Contact(in1 := "AI_AGTR3262_Toc_Do_AO", in2 := 0.0)
      { S7_GenerateENO := "TRUE" } Move(in := 0.0, out1 => "AI_AGTR3262_Toc_Do_AO")
   END_RUNG
   // the same network as SCL:
   IF "AI_AGTR3262_Toc_Do_AO" < 0.0 THEN "AI_AGTR3262_Toc_Do_AO" := 0.0; END_IF;
END_REGION

REGION Network 170: Clamp tốc độ cánh khuấy Bồn 3 trong dải 0.0-100.0 (Trên)
   RUNG wire#powerrail
      { S7_Templates := "SrcType := Real" } GT_Contact(in1 := "AI_AGTR3262_Toc_Do_AO", in2 := 100.0)
      { S7_GenerateENO := "TRUE" } Move(in := 100.0, out1 => "AI_AGTR3262_Toc_Do_AO")
   END_RUNG
   // the same network as SCL:
   IF "AI_AGTR3262_Toc_Do_AO" > 100.0 THEN "AI_AGTR3262_Toc_Do_AO" := 100.0; END_IF;
END_REGION

REGION Network 171: Reset CV hơi Bồn 4 khi không chạy PID
   RUNG wire#powerrail
      I_Contact( "AI_PID_Bon4_Enable" )
      { S7_GenerateENO := "TRUE" } Move(in := 0.0, out1 => "AI_CV3216_Hoi_Bon4")
   END_RUNG
   // the same network as SCL:
   IF NOT "AI_PID_Bon4_Enable" THEN "AI_CV3216_Hoi_Bon4" := 0.0; END_IF;
END_REGION

REGION Network 172: Reset CV hơi Bồn 4 khi Stop hoặc Lỗi tổng PLC2
   RUNG wire#powerrail
      Contact( "AI_PLC2_Stop_Active" )
      wire#w1
      { S7_GenerateENO := "TRUE" } Move(in := 0.0, out1 => "AI_CV3216_Hoi_Bon4")
   END_RUNG
   RUNG wire#powerrail
      Contact( "AI_PLC2_Loi_Tong" )
   END_RUNG wire#w1
   // the same network as SCL:
   IF "AI_PLC2_Stop_Active" OR "AI_PLC2_Loi_Tong" THEN "AI_CV3216_Hoi_Bon4" := 0.0; END_IF;
END_REGION

REGION Network 173: Clamp CV hơi Bồn 4 trong dải 0.0-100.0 (Dưới)
   RUNG wire#powerrail
      { S7_Templates := "SrcType := Real" } LT_Contact(in1 := "AI_CV3216_Hoi_Bon4", in2 := 0.0)
      { S7_GenerateENO := "TRUE" } Move(in := 0.0, out1 => "AI_CV3216_Hoi_Bon4")
   END_RUNG
   // the same network as SCL:
   IF "AI_CV3216_Hoi_Bon4" < 0.0 THEN "AI_CV3216_Hoi_Bon4" := 0.0; END_IF;
END_REGION

REGION Network 174: Clamp CV hơi Bồn 4 trong dải 0.0-100.0 (Trên)
   RUNG wire#powerrail
      { S7_Templates := "SrcType := Real" } GT_Contact(in1 := "AI_CV3216_Hoi_Bon4", in2 := 100.0)
      { S7_GenerateENO := "TRUE" } Move(in := 100.0, out1 => "AI_CV3216_Hoi_Bon4")
   END_RUNG
   // the same network as SCL:
   IF "AI_CV3216_Hoi_Bon4" > 100.0 THEN "AI_CV3216_Hoi_Bon4" := 100.0; END_IF;
END_REGION

REGION Network 175: Reset tốc độ động cơ khuấy Bồn 4 khi không chạy
   RUNG wire#powerrail
      I_Contact( "AI_AGTR3263_Khuay_Bon4" )
      { S7_GenerateENO := "TRUE" } Move(in := 0.0, out1 => "AI_AGTR3263_Toc_Do_AO")
   END_RUNG
   // the same network as SCL:
   IF NOT "AI_AGTR3263_Khuay_Bon4" THEN "AI_AGTR3263_Toc_Do_AO" := 0.0; END_IF;
END_REGION

REGION Network 176: Reset tốc độ động cơ khuấy Bồn 4 khi Stop hoặc Lỗi tổng PLC2
   RUNG wire#powerrail
      Contact( "AI_PLC2_Stop_Active" )
      wire#w1
      { S7_GenerateENO := "TRUE" } Move(in := 0.0, out1 => "AI_AGTR3263_Toc_Do_AO")
   END_RUNG
   RUNG wire#powerrail
      Contact( "AI_PLC2_Loi_Tong" )
   END_RUNG wire#w1
   // the same network as SCL:
   IF "AI_PLC2_Stop_Active" OR "AI_PLC2_Loi_Tong" THEN "AI_AGTR3263_Toc_Do_AO" := 0.0; END_IF;
END_REGION

REGION Network 177: Clamp tốc độ động cơ khuấy Bồn 4 trong dải 0.0-100.0 (Dưới)
   RUNG wire#powerrail
      { S7_Templates := "SrcType := Real" } LT_Contact(in1 := "AI_AGTR3263_Toc_Do_AO", in2 := 0.0)
      { S7_GenerateENO := "TRUE" } Move(in := 0.0, out1 => "AI_AGTR3263_Toc_Do_AO")
   END_RUNG
   // the same network as SCL:
   IF "AI_AGTR3263_Toc_Do_AO" < 0.0 THEN "AI_AGTR3263_Toc_Do_AO" := 0.0; END_IF;
END_REGION

REGION Network 178: Clamp tốc độ động cơ khuấy Bồn 4 trong dải 0.0-100.0 (Trên)
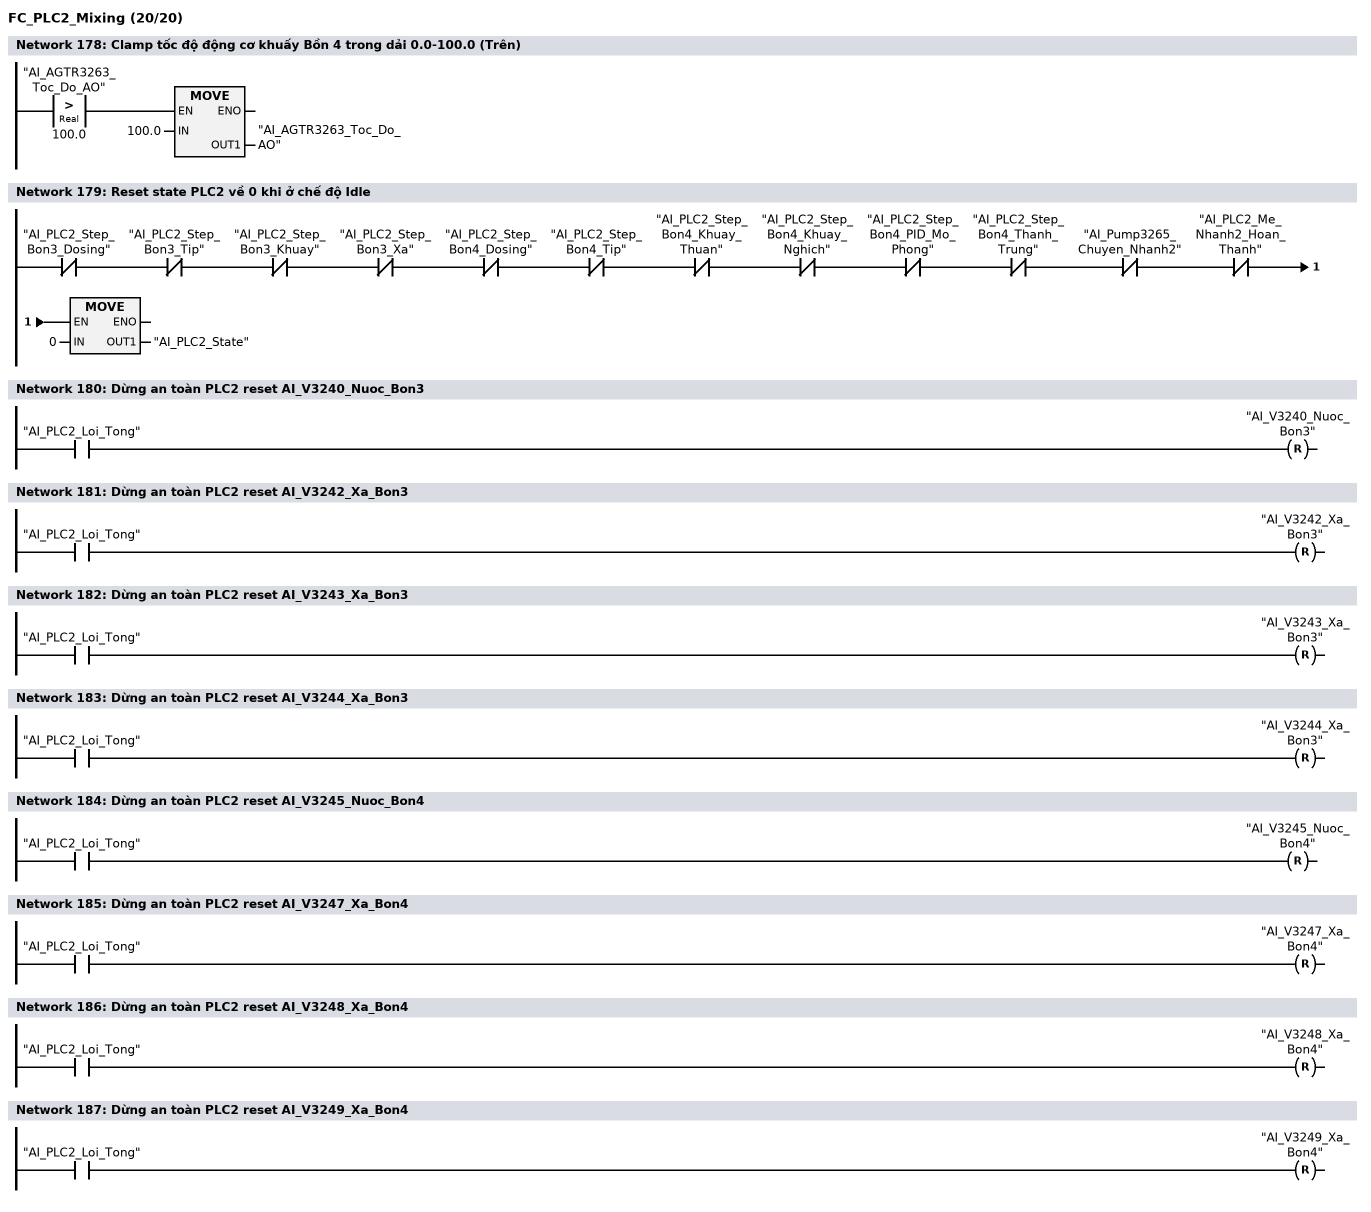
   RUNG wire#powerrail
      { S7_Templates := "SrcType := Real" } GT_Contact(in1 := "AI_AGTR3263_Toc_Do_AO", in2 := 100.0)
      { S7_GenerateENO := "TRUE" } Move(in := 100.0, out1 => "AI_AGTR3263_Toc_Do_AO")
   END_RUNG
   // the same network as SCL:
   IF "AI_AGTR3263_Toc_Do_AO" > 100.0 THEN "AI_AGTR3263_Toc_Do_AO" := 100.0; END_IF;
END_REGION

REGION Network 179: Reset state PLC2 về 0 khi ở chế độ Idle
   RUNG wire#powerrail
      I_Contact( "AI_PLC2_Step_Bon3_Dosing" )
      I_Contact( "AI_PLC2_Step_Bon3_Tip" )
      I_Contact( "AI_PLC2_Step_Bon3_Khuay" )
      I_Contact( "AI_PLC2_Step_Bon3_Xa" )
      I_Contact( "AI_PLC2_Step_Bon4_Dosing" )
      I_Contact( "AI_PLC2_Step_Bon4_Tip" )
      I_Contact( "AI_PLC2_Step_Bon4_Khuay_Thuan" )
      I_Contact( "AI_PLC2_Step_Bon4_Khuay_Nghich" )
      I_Contact( "AI_PLC2_Step_Bon4_PID_Mo_Phong" )
      I_Contact( "AI_PLC2_Step_Bon4_Thanh_Trung" )
      I_Contact( "AI_Pump3265_Chuyen_Nhanh2" )
      I_Contact( "AI_PLC2_Me_Nhanh2_Hoan_Thanh" )
      { S7_GenerateENO := "TRUE" } Move(in := 0, out1 => "AI_PLC2_State")
   END_RUNG
   // the same network as SCL:
   IF NOT "AI_PLC2_Step_Bon3_Dosing" AND NOT "AI_PLC2_Step_Bon3_Tip" AND NOT "AI_PLC2_Step_Bon3_Khuay" AND NOT "AI_PLC2_Step_Bon3_Xa" AND NOT "AI_PLC2_Step_Bon4_Dosing" AND NOT "AI_PLC2_Step_Bon4_Tip" AND NOT "AI_PLC2_Step_Bon4_Khuay_Thuan" AND NOT "AI_PLC2_Step_Bon4_Khuay_Nghich" AND NOT "AI_PLC2_Step_Bon4_PID_Mo_Phong" AND NOT "AI_PLC2_Step_Bon4_Thanh_Trung" AND NOT "AI_Pump3265_Chuyen_Nhanh2" AND NOT "AI_PLC2_Me_Nhanh2_Hoan_Thanh" THEN
       "AI_PLC2_State" := 0;
   END_IF;
END_REGION

REGION Network 180: Dừng an toàn PLC2 reset AI_V3240_Nuoc_Bon3
   RUNG wire#powerrail
      Contact( "AI_PLC2_Loi_Tong" )
      R_Coil( "AI_V3240_Nuoc_Bon3" )
   END_RUNG
   // the same network as SCL:
   IF "AI_PLC2_Loi_Tong" THEN "AI_V3240_Nuoc_Bon3" := FALSE; END_IF;
END_REGION

REGION Network 181: Dừng an toàn PLC2 reset AI_V3242_Xa_Bon3
   RUNG wire#powerrail
      Contact( "AI_PLC2_Loi_Tong" )
      R_Coil( "AI_V3242_Xa_Bon3" )
   END_RUNG
   // the same network as SCL:
   IF "AI_PLC2_Loi_Tong" THEN "AI_V3242_Xa_Bon3" := FALSE; END_IF;
END_REGION

REGION Network 182: Dừng an toàn PLC2 reset AI_V3243_Xa_Bon3
   RUNG wire#powerrail
      Contact( "AI_PLC2_Loi_Tong" )
      R_Coil( "AI_V3243_Xa_Bon3" )
   END_RUNG
   // the same network as SCL:
   IF "AI_PLC2_Loi_Tong" THEN "AI_V3243_Xa_Bon3" := FALSE; END_IF;
END_REGION

REGION Network 183: Dừng an toàn PLC2 reset AI_V3244_Xa_Bon3
   RUNG wire#powerrail
      Contact( "AI_PLC2_Loi_Tong" )
      R_Coil( "AI_V3244_Xa_Bon3" )
   END_RUNG
   // the same network as SCL:
   IF "AI_PLC2_Loi_Tong" THEN "AI_V3244_Xa_Bon3" := FALSE; END_IF;
END_REGION

REGION Network 184: Dừng an toàn PLC2 reset AI_V3245_Nuoc_Bon4
   RUNG wire#powerrail
      Contact( "AI_PLC2_Loi_Tong" )
      R_Coil( "AI_V3245_Nuoc_Bon4" )
   END_RUNG
   // the same network as SCL:
   IF "AI_PLC2_Loi_Tong" THEN "AI_V3245_Nuoc_Bon4" := FALSE; END_IF;
END_REGION

REGION Network 185: Dừng an toàn PLC2 reset AI_V3247_Xa_Bon4
   RUNG wire#powerrail
      Contact( "AI_PLC2_Loi_Tong" )
      R_Coil( "AI_V3247_Xa_Bon4" )
   END_RUNG
   // the same network as SCL:
   IF "AI_PLC2_Loi_Tong" THEN "AI_V3247_Xa_Bon4" := FALSE; END_IF;
END_REGION

REGION Network 186: Dừng an toàn PLC2 reset AI_V3248_Xa_Bon4
   RUNG wire#powerrail
      Contact( "AI_PLC2_Loi_Tong" )
      R_Coil( "AI_V3248_Xa_Bon4" )
   END_RUNG
   // the same network as SCL:
   IF "AI_PLC2_Loi_Tong" THEN "AI_V3248_Xa_Bon4" := FALSE; END_IF;
END_REGION

REGION Network 187: Dừng an toàn PLC2 reset AI_V3249_Xa_Bon4
   RUNG wire#powerrail
      Contact( "AI_PLC2_Loi_Tong" )
      R_Coil( "AI_V3249_Xa_Bon4" )
   END_RUNG
   // the same network as SCL:
   IF "AI_PLC2_Loi_Tong" THEN "AI_V3249_Xa_Bon4" := FALSE; END_IF;
END_REGION
END_FUNCTION

FUNCTION "FC_PLC1_Logic" : Void   // FC10, LAD
{ S7_Optimized_Access := 'TRUE' }
VERSION : 0.1
// stored: AutoNumber true, IsIECCheckEnabled false, SetENOAutomatically false, UDAEnableTagReadback false
BEGIN

REGION Network 1: Start Motor - Set bMotorRunning
